ABB RAPID module: Module1.mod

MODULE Module1

! ## =========================================================================== ##
    ! MIT License
    ! Copyright (c) 2021 Roman Parak
    ! Permission is hereby granted, free of charge, to any person obtaining a copy
    ! of this software and associated documentation files (the "Software"), to deal
    ! in the Software without restriction, including without limitation the rights
    ! to use, copy, modify, merge, publish, distribute, sublicense, and/or sell
    ! copies of the Software, and to permit persons to whom the Software is
    ! furnished to do so, subject to the following conditions:
    ! The above copyright notice and this permission notice shall be included in all
    ! copies or substantial portions of the Software.
    ! THE SOFTWARE IS PROVIDED "AS IS", WITHOUT WARRANTY OF ANY KIND, EXPRESS OR
    ! IMPLIED, INCLUDING BUT NOT LIMITED TO THE WARRANTIES OF MERCHANTABILITY,
    ! FITNESS FOR A PARTICULAR PURPOSE AND NONINFRINGEMENT. IN NO EVENT SHALL THE
    ! AUTHORS OR COPYRIGHT HOLDERS BE LIABLE FOR ANY CLAIM, DAMAGES OR OTHER
    ! LIABILITY, WHETHER IN AN ACTION OF CONTRACT, TORT OR OTHERWISE, ARISING FROM,
    ! OUT OF OR IN CONNECTION WITH THE SOFTWARE OR THE USE OR OTHER DEALINGS IN THE
    ! SOFTWARE.
    ! ## =========================================================================== ##
    ! Author   : Roman Parak
    ! Email    : Roman.Parak@outlook.com
    ! Github   : https://github.com/rparak
    ! File Name: T_ROB1/Module1.mod
    ! ## =========================================================================== ##

    ! ############### EGM Initialization Parameters ############### !
    ! Identifier for the EGM correction.
     VAR robtarget starting_position;

    ! ################################## Externally Guided motion (EGM) - Main Cycle ################################## !
    PROC main()
        starting_position := CRobT(\Tool:=Tooldata_7\wobj:=wobj0);
        ConfJ\Off;
MoveJ RelTool (starting_position, 198, 1.3, -561 \Rx:=3.2, \Ry:=11.1, \Rz:=0), v200, z200, Tooldata_7;
MoveJ RelTool (starting_position, 198, 1.5, -561 \Rx:=3.1, \Ry:=11.1, \Rz:=0), v200, z200, Tooldata_7;
MoveJ RelTool (starting_position, 198, 1.7, -562 \Rx:=3, \Ry:=11.1, \Rz:=0), v200, z200, Tooldata_7;
MoveJ RelTool (starting_position, 198, 1.9, -562 \Rx:=2.8, \Ry:=11.1, \Rz:=0), v200, z200, Tooldata_7;
MoveJ RelTool (starting_position, 198, 2.1, -563 \Rx:=2.7, \Ry:=11.1, \Rz:=0), v200, z200, Tooldata_7;
MoveJ RelTool (starting_position, 198, 2.3, -563 \Rx:=2.6, \Ry:=11.1, \Rz:=0), v200, z200, Tooldata_7;
MoveJ RelTool (starting_position, 198, 2.6, -564 \Rx:=2.5, \Ry:=11.1, \Rz:=0), v200, z200, Tooldata_7;
MoveJ RelTool (starting_position, 197, 2.9, -565 \Rx:=2.3, \Ry:=11.1, \Rz:=0), v200, z200, Tooldata_7;
MoveJ RelTool (starting_position, 197, 3.1, -565 \Rx:=2.2, \Ry:=11.1, \Rz:=0), v200, z200, Tooldata_7;
MoveJ RelTool (starting_position, 197, 3.5, -566 \Rx:=2.1, \Ry:=10.8, \Rz:=0), v200, z200, Tooldata_7;
MoveJ RelTool (starting_position, 196, 3.8, -567 \Rx:=2, \Ry:=10.8, \Rz:=0), v200, z200, Tooldata_7;
MoveJ RelTool (starting_position, 196, 4.1, -567 \Rx:=2, \Ry:=10.8, \Rz:=0), v200, z200, Tooldata_7;
MoveJ RelTool (starting_position, 195, 4.5, -568 \Rx:=1.9, \Ry:=10.5, \Rz:=0), v200, z200, Tooldata_7;
MoveJ RelTool (starting_position, 195, 4.9, -569 \Rx:=1.9, \Ry:=10.5, \Rz:=0), v200, z200, Tooldata_7;
MoveJ RelTool (starting_position, 194, 5.3, -570 \Rx:=1.8, \Ry:=10.5, \Rz:=0), v200, z200, Tooldata_7;
MoveJ RelTool (starting_position, 194, 5.8, -571 \Rx:=1.8, \Ry:=10.5, \Rz:=0), v200, z200, Tooldata_7;
MoveJ RelTool (starting_position, 193, 6.3, -572 \Rx:=1.7, \Ry:=10.2, \Rz:=0), v200, z200, Tooldata_7;
MoveJ RelTool (starting_position, 192, 6.7, -573 \Rx:=1.7, \Ry:=10.2, \Rz:=0), v200, z200, Tooldata_7;
MoveJ RelTool (starting_position, 191, 7.3, -574 \Rx:=1.6, \Ry:=9.9, \Rz:=0), v200, z200, Tooldata_7;
MoveJ RelTool (starting_position, 190, 7.8, -575 \Rx:=1.6, \Ry:=9.9, \Rz:=0), v200, z200, Tooldata_7;
MoveJ RelTool (starting_position, 190, 8.4, -576 \Rx:=1.6, \Ry:=9.6, \Rz:=0), v200, z200, Tooldata_7;
MoveJ RelTool (starting_position, 189, 8.9, -577 \Rx:=1.5, \Ry:=9.6, \Rz:=0), v200, z200, Tooldata_7;
MoveJ RelTool (starting_position, 188, 9.6, -578 \Rx:=1.5, \Ry:=9.3, \Rz:=0), v200, z200, Tooldata_7;
MoveJ RelTool (starting_position, 187, 10.2, -579 \Rx:=1.5, \Ry:=9.3, \Rz:=0), v200, z200, Tooldata_7;
MoveJ RelTool (starting_position, 186, 10.8, -580 \Rx:=1.5, \Ry:=9, \Rz:=0), v200, z200, Tooldata_7;
MoveJ RelTool (starting_position, 185, 11.5, -581 \Rx:=1.5, \Ry:=8.7, \Rz:=0), v200, z200, Tooldata_7;
MoveJ RelTool (starting_position, 183, 12.1, -582 \Rx:=1.5, \Ry:=8.7, \Rz:=0), v200, z200, Tooldata_7;
MoveJ RelTool (starting_position, 182, 12.8, -583 \Rx:=1.5, \Ry:=8.4, \Rz:=0), v200, z200, Tooldata_7;
MoveJ RelTool (starting_position, 181, 13.5, -584 \Rx:=1.5, \Ry:=8.1, \Rz:=0), v200, z200, Tooldata_7;
MoveJ RelTool (starting_position, 179, 14.2, -585 \Rx:=1.5, \Ry:=7.8, \Rz:=0), v200, z200, Tooldata_7;
MoveJ RelTool (starting_position, 178, 14.9, -586 \Rx:=1.5, \Ry:=7.8, \Rz:=0), v200, z200, Tooldata_7;
MoveJ RelTool (starting_position, 177, 15.7, -586 \Rx:=1.5, \Ry:=7.5, \Rz:=0), v200, z200, Tooldata_7;
MoveJ RelTool (starting_position, 175, 16.4, -587 \Rx:=1.4, \Ry:=7.2, \Rz:=0), v200, z200, Tooldata_7;
MoveJ RelTool (starting_position, 174, 17.1, -588 \Rx:=1.4, \Ry:=6.9, \Rz:=0), v200, z200, Tooldata_7;
MoveJ RelTool (starting_position, 172, 17.8, -589 \Rx:=1.3, \Ry:=6.6, \Rz:=0), v200, z200, Tooldata_7;
MoveJ RelTool (starting_position, 171, 18.5, -589 \Rx:=1.3, \Ry:=6.3, \Rz:=0), v200, z200, Tooldata_7;
MoveJ RelTool (starting_position, 169, 19.2, -590 \Rx:=1.2, \Ry:=6, \Rz:=0), v200, z200, Tooldata_7;
MoveJ RelTool (starting_position, 168, 19.9, -591 \Rx:=1.1, \Ry:=6, \Rz:=0), v200, z200, Tooldata_7;
MoveJ RelTool (starting_position, 166, 20.5, -591 \Rx:=1, \Ry:=5.7, \Rz:=0), v200, z200, Tooldata_7;
MoveJ RelTool (starting_position, 165, 21.2, -592 \Rx:=0.9, \Ry:=5.4, \Rz:=0), v200, z200, Tooldata_7;
MoveJ RelTool (starting_position, 163, 21.8, -592 \Rx:=0.7, \Ry:=5.1, \Rz:=0), v200, z200, Tooldata_7;
MoveJ RelTool (starting_position, 162, 22.4, -593 \Rx:=0.6, \Ry:=4.8, \Rz:=0), v200, z200, Tooldata_7;
MoveJ RelTool (starting_position, 160, 23, -593 \Rx:=0.5, \Ry:=4.5, \Rz:=0), v200, z200, Tooldata_7;
MoveJ RelTool (starting_position, 158, 23.6, -594 \Rx:=0.4, \Ry:=4.2, \Rz:=0), v200, z200, Tooldata_7;
MoveJ RelTool (starting_position, 157, 24.1, -594 \Rx:=0.2, \Ry:=3.9, \Rz:=0), v200, z200, Tooldata_7;
MoveJ RelTool (starting_position, 155, 24.6, -594 \Rx:=0.1, \Ry:=3.6, \Rz:=0), v200, z200, Tooldata_7;
MoveJ RelTool (starting_position, 154, 25.1, -595 \Rx:=-0, \Ry:=3.6, \Rz:=0), v200, z200, Tooldata_7;
MoveJ RelTool (starting_position, 153, 25.6, -595 \Rx:=-0.1, \Ry:=3.3, \Rz:=0), v200, z200, Tooldata_7;
MoveJ RelTool (starting_position, 152, 26, -595 \Rx:=-0.1, \Ry:=3, \Rz:=0), v200, z200, Tooldata_7;
MoveJ RelTool (starting_position, 151, 26.4, -595 \Rx:=-0.2, \Ry:=3, \Rz:=0), v200, z200, Tooldata_7;
MoveJ RelTool (starting_position, 150, 26.8, -595 \Rx:=-0.3, \Ry:=2.7, \Rz:=0), v200, z200, Tooldata_7;
MoveJ RelTool (starting_position, 149, 27.1, -596 \Rx:=-0.3, \Ry:=2.7, \Rz:=0), v200, z200, Tooldata_7;
MoveJ RelTool (starting_position, 148, 27.5, -596 \Rx:=-0.3, \Ry:=2.4, \Rz:=0), v200, z200, Tooldata_7;
MoveJ RelTool (starting_position, 147, 27.8, -596 \Rx:=-0.3, \Ry:=2.1, \Rz:=0), v200, z200, Tooldata_7;
MoveJ RelTool (starting_position, 146, 28.2, -596 \Rx:=-0.3, \Ry:=2.1, \Rz:=0), v200, z200, Tooldata_7;
MoveJ RelTool (starting_position, 146, 28.5, -596 \Rx:=-0.3, \Ry:=2.1, \Rz:=0), v200, z200, Tooldata_7;
MoveJ RelTool (starting_position, 145, 28.8, -596 \Rx:=-0.3, \Ry:=2.1, \Rz:=0), v200, z200, Tooldata_7;
MoveJ RelTool (starting_position, 145, 29, -596 \Rx:=-0.2, \Ry:=1.8, \Rz:=0), v200, z200, Tooldata_7;
MoveJ RelTool (starting_position, 145, 29.3, -596 \Rx:=-0.1, \Ry:=1.8, \Rz:=0), v200, z200, Tooldata_7;
MoveJ RelTool (starting_position, 144, 29.6, -596 \Rx:=0, \Ry:=1.8, \Rz:=0), v200, z200, Tooldata_7;
MoveJ RelTool (starting_position, 144, 29.8, -596 \Rx:=0.1, \Ry:=1.8, \Rz:=0), v200, z200, Tooldata_7;
MoveJ RelTool (starting_position, 144, 30.1, -597 \Rx:=0.3, \Ry:=1.8, \Rz:=0), v200, z200, Tooldata_7;
MoveJ RelTool (starting_position, 144, 30.4, -597 \Rx:=0.4, \Ry:=1.8, \Rz:=0), v200, z200, Tooldata_7;
MoveJ RelTool (starting_position, 144, 30.6, -597 \Rx:=0.6, \Ry:=1.8, \Rz:=0), v200, z200, Tooldata_7;
MoveJ RelTool (starting_position, 144, 30.9, -597 \Rx:=0.8, \Ry:=1.8, \Rz:=0), v200, z200, Tooldata_7;
MoveJ RelTool (starting_position, 144, 31.2, -597 \Rx:=0.9, \Ry:=1.8, \Rz:=0), v200, z200, Tooldata_7;
MoveJ RelTool (starting_position, 144, 31.5, -597 \Rx:=1.2, \Ry:=1.8, \Rz:=0), v200, z200, Tooldata_7;
MoveJ RelTool (starting_position, 144, 31.8, -597 \Rx:=1.4, \Ry:=1.8, \Rz:=0), v200, z200, Tooldata_7;
MoveJ RelTool (starting_position, 144, 32.1, -597 \Rx:=1.7, \Ry:=1.8, \Rz:=0), v200, z200, Tooldata_7;
MoveJ RelTool (starting_position, 145, 32.4, -597 \Rx:=2, \Ry:=1.8, \Rz:=0), v200, z200, Tooldata_7;
MoveJ RelTool (starting_position, 145, 32.8, -597 \Rx:=2.4, \Ry:=1.8, \Rz:=0), v200, z200, Tooldata_7;
MoveJ RelTool (starting_position, 145, 33.2, -597 \Rx:=2.7, \Ry:=2.1, \Rz:=0), v200, z200, Tooldata_7;
MoveJ RelTool (starting_position, 146, 33.6, -597 \Rx:=3.1, \Ry:=2.1, \Rz:=0), v200, z200, Tooldata_7;
MoveJ RelTool (starting_position, 146, 34, -598 \Rx:=3.4, \Ry:=2.1, \Rz:=0), v200, z200, Tooldata_7;
MoveJ RelTool (starting_position, 147, 34.4, -598 \Rx:=3.7, \Ry:=2.4, \Rz:=0), v200, z200, Tooldata_7;
MoveJ RelTool (starting_position, 147, 34.8, -598 \Rx:=4.1, \Ry:=2.4, \Rz:=0), v200, z200, Tooldata_7;
MoveJ RelTool (starting_position, 148, 35.3, -598 \Rx:=4.4, \Ry:=2.4, \Rz:=0), v200, z200, Tooldata_7;
MoveJ RelTool (starting_position, 148, 35.9, -598 \Rx:=4.7, \Ry:=2.4, \Rz:=0), v200, z200, Tooldata_7;
MoveJ RelTool (starting_position, 149, 36.4, -599 \Rx:=5, \Ry:=2.7, \Rz:=0), v200, z200, Tooldata_7;
MoveJ RelTool (starting_position, 149, 37, -599 \Rx:=5.3, \Ry:=2.7, \Rz:=0), v200, z200, Tooldata_7;
MoveJ RelTool (starting_position, 150, 37.6, -599 \Rx:=5.6, \Ry:=2.7, \Rz:=0), v200, z200, Tooldata_7;
MoveJ RelTool (starting_position, 150, 38.2, -600 \Rx:=5.8, \Ry:=3, \Rz:=0), v200, z200, Tooldata_7;
MoveJ RelTool (starting_position, 151, 38.8, -600 \Rx:=5.9, \Ry:=3, \Rz:=0), v200, z200, Tooldata_7;
MoveJ RelTool (starting_position, 151, 39.5, -600 \Rx:=6.1, \Ry:=3, \Rz:=0), v200, z200, Tooldata_7;
MoveJ RelTool (starting_position, 151, 40.2, -601 \Rx:=6.2, \Ry:=3, \Rz:=0), v200, z200, Tooldata_7;
MoveJ RelTool (starting_position, 151, 40.9, -601 \Rx:=6.3, \Ry:=3, \Rz:=0), v200, z200, Tooldata_7;
MoveJ RelTool (starting_position, 152, 41.6, -602 \Rx:=6.3, \Ry:=3, \Rz:=0), v200, z200, Tooldata_7;
MoveJ RelTool (starting_position, 152, 42.4, -602 \Rx:=6.2, \Ry:=3.3, \Rz:=0), v200, z200, Tooldata_7;
MoveJ RelTool (starting_position, 152, 43.1, -603 \Rx:=6.2, \Ry:=3.3, \Rz:=0), v200, z200, Tooldata_7;
MoveJ RelTool (starting_position, 153, 43.8, -603 \Rx:=6, \Ry:=3.3, \Rz:=0), v200, z200, Tooldata_7;
MoveJ RelTool (starting_position, 153, 44.6, -604 \Rx:=5.9, \Ry:=3.3, \Rz:=0), v200, z200, Tooldata_7;
MoveJ RelTool (starting_position, 153, 45.4, -604 \Rx:=5.7, \Ry:=3.3, \Rz:=0), v200, z200, Tooldata_7;
MoveJ RelTool (starting_position, 153, 46.1, -605 \Rx:=5.6, \Ry:=3.6, \Rz:=0), v200, z200, Tooldata_7;
MoveJ RelTool (starting_position, 153, 46.9, -605 \Rx:=5.3, \Ry:=3.3, \Rz:=0), v200, z200, Tooldata_7;
MoveJ RelTool (starting_position, 153, 47.6, -606 \Rx:=5.1, \Ry:=3.3, \Rz:=0), v200, z200, Tooldata_7;
MoveJ RelTool (starting_position, 153, 48.3, -606 \Rx:=4.9, \Ry:=3.3, \Rz:=0), v200, z200, Tooldata_7;
MoveJ RelTool (starting_position, 152, 49.1, -606 \Rx:=4.7, \Ry:=3.3, \Rz:=0), v200, z200, Tooldata_7;
MoveJ RelTool (starting_position, 152, 49.8, -607 \Rx:=4.5, \Ry:=3.3, \Rz:=0), v200, z200, Tooldata_7;
MoveJ RelTool (starting_position, 152, 50.5, -607 \Rx:=4.2, \Ry:=3, \Rz:=0), v200, z200, Tooldata_7;
MoveJ RelTool (starting_position, 151, 51.1, -608 \Rx:=4, \Ry:=3, \Rz:=0), v200, z200, Tooldata_7;
MoveJ RelTool (starting_position, 151, 51.8, -608 \Rx:=3.9, \Ry:=3, \Rz:=0), v200, z200, Tooldata_7;
MoveJ RelTool (starting_position, 151, 52.4, -608 \Rx:=3.7, \Ry:=3, \Rz:=0), v200, z200, Tooldata_7;
MoveJ RelTool (starting_position, 150, 53, -609 \Rx:=3.6, \Ry:=3, \Rz:=0), v200, z200, Tooldata_7;
MoveJ RelTool (starting_position, 150, 53.6, -609 \Rx:=3.5, \Ry:=2.7, \Rz:=0), v200, z200, Tooldata_7;
MoveJ RelTool (starting_position, 150, 54.1, -609 \Rx:=3.4, \Ry:=2.7, \Rz:=0), v200, z200, Tooldata_7;
MoveJ RelTool (starting_position, 149, 54.6, -609 \Rx:=3.4, \Ry:=2.7, \Rz:=0), v200, z200, Tooldata_7;
MoveJ RelTool (starting_position, 149, 55.1, -610 \Rx:=3.3, \Ry:=2.7, \Rz:=0), v200, z200, Tooldata_7;
MoveJ RelTool (starting_position, 148, 55.6, -610 \Rx:=3.3, \Ry:=2.4, \Rz:=0), v200, z200, Tooldata_7;
MoveJ RelTool (starting_position, 148, 56, -610 \Rx:=3.4, \Ry:=2.4, \Rz:=0), v200, z200, Tooldata_7;
MoveJ RelTool (starting_position, 147, 56.4, -610 \Rx:=3.4, \Ry:=2.4, \Rz:=0), v200, z200, Tooldata_7;
MoveJ RelTool (starting_position, 147, 56.8, -610 \Rx:=3.6, \Ry:=2.1, \Rz:=0), v200, z200, Tooldata_7;
MoveJ RelTool (starting_position, 146, 57.1, -610 \Rx:=3.7, \Ry:=2.1, \Rz:=0), v200, z200, Tooldata_7;
MoveJ RelTool (starting_position, 146, 57.5, -611 \Rx:=4, \Ry:=2.1, \Rz:=0), v200, z200, Tooldata_7;
MoveJ RelTool (starting_position, 145, 57.8, -611 \Rx:=4.2, \Ry:=2.1, \Rz:=0), v200, z200, Tooldata_7;
MoveJ RelTool (starting_position, 145, 58.1, -611 \Rx:=4.6, \Ry:=1.8, \Rz:=0), v200, z200, Tooldata_7;
MoveJ RelTool (starting_position, 144, 58.4, -611 \Rx:=5, \Ry:=1.8, \Rz:=0), v200, z200, Tooldata_7;
MoveJ RelTool (starting_position, 144, 58.7, -611 \Rx:=5.4, \Ry:=1.8, \Rz:=0), v200, z200, Tooldata_7;
MoveJ RelTool (starting_position, 143, 59, -612 \Rx:=5.8, \Ry:=1.5, \Rz:=0), v200, z200, Tooldata_7;
MoveJ RelTool (starting_position, 142, 59.2, -612 \Rx:=6.2, \Ry:=1.5, \Rz:=0), v200, z200, Tooldata_7;
MoveJ RelTool (starting_position, 142, 59.5, -612 \Rx:=6.6, \Ry:=1.5, \Rz:=0), v200, z200, Tooldata_7;
MoveJ RelTool (starting_position, 141, 59.7, -612 \Rx:=7.1, \Ry:=1.2, \Rz:=0), v200, z200, Tooldata_7;
MoveJ RelTool (starting_position, 140, 60, -612 \Rx:=7.6, \Ry:=1.2, \Rz:=0), v200, z200, Tooldata_7;
MoveJ RelTool (starting_position, 139, 60.2, -613 \Rx:=8.1, \Ry:=0.9, \Rz:=0), v200, z200, Tooldata_7;
MoveJ RelTool (starting_position, 139, 60.5, -613 \Rx:=8.5, \Ry:=0.9, \Rz:=0), v200, z200, Tooldata_7;
MoveJ RelTool (starting_position, 138, 60.7, -613 \Rx:=9, \Ry:=0.6, \Rz:=0), v200, z200, Tooldata_7;
MoveJ RelTool (starting_position, 137, 61, -613 \Rx:=9.4, \Ry:=0.6, \Rz:=0), v200, z200, Tooldata_7;
MoveJ RelTool (starting_position, 136, 61.2, -613 \Rx:=9.8, \Ry:=0.6, \Rz:=0), v200, z200, Tooldata_7;
MoveJ RelTool (starting_position, 135, 61.5, -614 \Rx:=10.1, \Ry:=0.3, \Rz:=0), v200, z200, Tooldata_7;
MoveJ RelTool (starting_position, 134, 61.8, -614 \Rx:=10.3, \Ry:=0, \Rz:=0), v200, z200, Tooldata_7;
MoveJ RelTool (starting_position, 133, 62.1, -614 \Rx:=10.5, \Ry:=-0, \Rz:=0), v200, z200, Tooldata_7;
MoveJ RelTool (starting_position, 133, 62.5, -614 \Rx:=10.6, \Ry:=-0.3, \Rz:=0), v200, z200, Tooldata_7;
MoveJ RelTool (starting_position, 132, 62.8, -614 \Rx:=10.6, \Ry:=-0.3, \Rz:=0), v200, z200, Tooldata_7;
MoveJ RelTool (starting_position, 131, 63.2, -614 \Rx:=10.6, \Ry:=-0.6, \Rz:=0), v200, z200, Tooldata_7;
MoveJ RelTool (starting_position, 130, 63.6, -614 \Rx:=10.4, \Ry:=-0.6, \Rz:=0), v200, z200, Tooldata_7;
MoveJ RelTool (starting_position, 129, 64, -614 \Rx:=10.1, \Ry:=-0.9, \Rz:=0), v200, z200, Tooldata_7;
MoveJ RelTool (starting_position, 128, 64.4, -614 \Rx:=9.8, \Ry:=-1.2, \Rz:=0), v200, z200, Tooldata_7;
MoveJ RelTool (starting_position, 127, 64.8, -614 \Rx:=9.5, \Ry:=-1.2, \Rz:=0), v200, z200, Tooldata_7;
MoveJ RelTool (starting_position, 126, 65.3, -614 \Rx:=9.1, \Ry:=-1.5, \Rz:=0), v200, z200, Tooldata_7;
MoveJ RelTool (starting_position, 125, 65.9, -613 \Rx:=8.7, \Ry:=-1.5, \Rz:=0), v200, z200, Tooldata_7;
MoveJ RelTool (starting_position, 124, 66.4, -613 \Rx:=8.2, \Ry:=-1.8, \Rz:=0), v200, z200, Tooldata_7;
MoveJ RelTool (starting_position, 123, 67, -613 \Rx:=7.7, \Ry:=-1.8, \Rz:=0), v200, z200, Tooldata_7;
MoveJ RelTool (starting_position, 122, 67.6, -613 \Rx:=7.2, \Ry:=-2.1, \Rz:=0), v200, z200, Tooldata_7;
MoveJ RelTool (starting_position, 122, 68.2, -612 \Rx:=6.7, \Ry:=-2.1, \Rz:=0), v200, z200, Tooldata_7;
MoveJ RelTool (starting_position, 121, 68.8, -612 \Rx:=6.2, \Ry:=-2.1, \Rz:=0), v200, z200, Tooldata_7;
MoveJ RelTool (starting_position, 120, 69.5, -612 \Rx:=5.7, \Ry:=-2.4, \Rz:=0), v200, z200, Tooldata_7;
MoveJ RelTool (starting_position, 119, 70.2, -611 \Rx:=5.2, \Ry:=-2.7, \Rz:=0), v200, z200, Tooldata_7;
MoveJ RelTool (starting_position, 118, 70.9, -611 \Rx:=4.8, \Ry:=-2.7, \Rz:=0), v200, z200, Tooldata_7;
MoveJ RelTool (starting_position, 117, 71.6, -611 \Rx:=4.4, \Ry:=-3, \Rz:=0), v200, z200, Tooldata_7;
MoveJ RelTool (starting_position, 116, 72.4, -610 \Rx:=4.1, \Ry:=-3, \Rz:=0), v200, z200, Tooldata_7;
MoveJ RelTool (starting_position, 116, 73.1, -610 \Rx:=3.8, \Ry:=-3, \Rz:=0), v200, z200, Tooldata_7;
MoveJ RelTool (starting_position, 115, 73.8, -610 \Rx:=3.5, \Ry:=-3.3, \Rz:=0), v200, z200, Tooldata_7;
MoveJ RelTool (starting_position, 114, 74.6, -609 \Rx:=3.3, \Ry:=-3.3, \Rz:=0), v200, z200, Tooldata_7;
MoveJ RelTool (starting_position, 114, 75.4, -609 \Rx:=3.1, \Ry:=-3.6, \Rz:=0), v200, z200, Tooldata_7;
MoveJ RelTool (starting_position, 113, 76.1, -608 \Rx:=3, \Ry:=-3.6, \Rz:=0), v200, z200, Tooldata_7;
MoveJ RelTool (starting_position, 113, 76.9, -608 \Rx:=3, \Ry:=-3.6, \Rz:=0), v200, z200, Tooldata_7;
MoveJ RelTool (starting_position, 113, 77.6, -608 \Rx:=2.9, \Ry:=-3.6, \Rz:=0), v200, z200, Tooldata_7;
MoveJ RelTool (starting_position, 112, 78.3, -607 \Rx:=2.9, \Ry:=-3.6, \Rz:=0), v200, z200, Tooldata_7;
MoveJ RelTool (starting_position, 112, 79.1, -607 \Rx:=2.9, \Ry:=-3.9, \Rz:=0), v200, z200, Tooldata_7;
MoveJ RelTool (starting_position, 111, 79.8, -606 \Rx:=2.9, \Ry:=-3.9, \Rz:=0), v200, z200, Tooldata_7;
MoveJ RelTool (starting_position, 111, 80.5, -606 \Rx:=3, \Ry:=-3.9, \Rz:=0), v200, z200, Tooldata_7;
MoveJ RelTool (starting_position, 110, 81.1, -605 \Rx:=3.1, \Ry:=-4.2, \Rz:=0), v200, z200, Tooldata_7;
MoveJ RelTool (starting_position, 110, 81.8, -605 \Rx:=3.1, \Ry:=-4.2, \Rz:=0), v200, z200, Tooldata_7;
MoveJ RelTool (starting_position, 110, 82.4, -605 \Rx:=3.2, \Ry:=-4.2, \Rz:=0), v200, z200, Tooldata_7;
MoveJ RelTool (starting_position, 109, 83, -604 \Rx:=3.2, \Ry:=-4.2, \Rz:=0), v200, z200, Tooldata_7;
MoveJ RelTool (starting_position, 109, 83.6, -604 \Rx:=3.2, \Ry:=-4.2, \Rz:=0), v200, z200, Tooldata_7;
MoveJ RelTool (starting_position, 108, 84.1, -603 \Rx:=3.3, \Ry:=-4.5, \Rz:=0), v200, z200, Tooldata_7;
MoveJ RelTool (starting_position, 108, 84.6, -603 \Rx:=3.3, \Ry:=-4.5, \Rz:=0), v200, z200, Tooldata_7;
MoveJ RelTool (starting_position, 108, 85.1, -602 \Rx:=3.3, \Ry:=-4.5, \Rz:=0), v200, z200, Tooldata_7;
MoveJ RelTool (starting_position, 107, 85.6, -602 \Rx:=3.3, \Ry:=-4.5, \Rz:=0), v200, z200, Tooldata_7;
MoveJ RelTool (starting_position, 107, 86, -602 \Rx:=3.3, \Ry:=-4.8, \Rz:=0), v200, z200, Tooldata_7;
MoveJ RelTool (starting_position, 106, 86.4, -601 \Rx:=3.3, \Ry:=-4.8, \Rz:=0), v200, z200, Tooldata_7;
MoveJ RelTool (starting_position, 106, 86.8, -601 \Rx:=3.2, \Ry:=-4.8, \Rz:=0), v200, z200, Tooldata_7;
MoveJ RelTool (starting_position, 106, 87.1, -600 \Rx:=3.2, \Ry:=-4.8, \Rz:=0), v200, z200, Tooldata_7;
MoveJ RelTool (starting_position, 106, 87.5, -600 \Rx:=3.2, \Ry:=-4.8, \Rz:=0), v200, z200, Tooldata_7;
MoveJ RelTool (starting_position, 106, 87.7, -600 \Rx:=3.1, \Ry:=-4.8, \Rz:=0), v200, z200, Tooldata_7;
MoveJ RelTool (starting_position, 105, 88, -599 \Rx:=3.1, \Ry:=-5.1, \Rz:=0), v200, z200, Tooldata_7;
MoveJ RelTool (starting_position, 105, 88.3, -599 \Rx:=3.1, \Ry:=-5.1, \Rz:=0), v200, z200, Tooldata_7;
MoveJ RelTool (starting_position, 105, 88.6, -598 \Rx:=3, \Ry:=-4.8, \Rz:=0), v200, z200, Tooldata_7;
MoveJ RelTool (starting_position, 105, 88.8, -598 \Rx:=3, \Ry:=-4.8, \Rz:=0), v200, z200, Tooldata_7;
MoveJ RelTool (starting_position, 105, 89.1, -597 \Rx:=3, \Ry:=-5.1, \Rz:=0), v200, z200, Tooldata_7;
MoveJ RelTool (starting_position, 105, 89.3, -597 \Rx:=3, \Ry:=-5.1, \Rz:=0), v200, z200, Tooldata_7;
MoveJ RelTool (starting_position, 104, 89.5, -596 \Rx:=2.9, \Ry:=-5.1, \Rz:=0), v200, z200, Tooldata_7;
MoveJ RelTool (starting_position, 104, 89.7, -595 \Rx:=2.9, \Ry:=-5.1, \Rz:=0), v200, z200, Tooldata_7;
MoveJ RelTool (starting_position, 104, 90, -595 \Rx:=2.8, \Ry:=-5.1, \Rz:=0), v200, z200, Tooldata_7;
MoveJ RelTool (starting_position, 105, 90.2, -594 \Rx:=2.7, \Ry:=-5.1, \Rz:=0), v200, z200, Tooldata_7;
MoveJ RelTool (starting_position, 105, 90.4, -594 \Rx:=2.6, \Ry:=-5.1, \Rz:=0), v200, z200, Tooldata_7;
MoveJ RelTool (starting_position, 105, 90.6, -593 \Rx:=2.4, \Ry:=-4.8, \Rz:=0), v200, z200, Tooldata_7;
MoveJ RelTool (starting_position, 106, 90.9, -592 \Rx:=2.3, \Ry:=-4.8, \Rz:=0), v200, z200, Tooldata_7;
MoveJ RelTool (starting_position, 106, 91.1, -592 \Rx:=2.1, \Ry:=-4.8, \Rz:=0), v200, z200, Tooldata_7;
MoveJ RelTool (starting_position, 107, 91.4, -591 \Rx:=1.9, \Ry:=-4.8, \Rz:=0), v200, z200, Tooldata_7;
MoveJ RelTool (starting_position, 107, 91.6, -590 \Rx:=1.7, \Ry:=-4.5, \Rz:=0), v200, z200, Tooldata_7;
MoveJ RelTool (starting_position, 108, 91.9, -590 \Rx:=1.5, \Ry:=-4.5, \Rz:=0), v200, z200, Tooldata_7;
MoveJ RelTool (starting_position, 108, 92.2, -589 \Rx:=1.3, \Ry:=-4.5, \Rz:=0), v200, z200, Tooldata_7;
MoveJ RelTool (starting_position, 109, 92.5, -588 \Rx:=1.1, \Ry:=-4.2, \Rz:=0), v200, z200, Tooldata_7;
MoveJ RelTool (starting_position, 110, 92.8, -588 \Rx:=0.9, \Ry:=-4.2, \Rz:=0), v200, z200, Tooldata_7;
MoveJ RelTool (starting_position, 111, 93.2, -587 \Rx:=0.7, \Ry:=-3.9, \Rz:=0), v200, z200, Tooldata_7;
MoveJ RelTool (starting_position, 112, 93.6, -587 \Rx:=0.4, \Ry:=-3.9, \Rz:=0), v200, z200, Tooldata_7;
MoveJ RelTool (starting_position, 113, 94, -586 \Rx:=0.2, \Ry:=-3.6, \Rz:=0), v200, z200, Tooldata_7;
MoveJ RelTool (starting_position, 114, 94.4, -586 \Rx:=0, \Ry:=-3.6, \Rz:=0), v200, z200, Tooldata_7;
MoveJ RelTool (starting_position, 115, 94.8, -585 \Rx:=-0.2, \Ry:=-3.3, \Rz:=0), v200, z200, Tooldata_7;
MoveJ RelTool (starting_position, 116, 95.3, -585 \Rx:=-0.4, \Ry:=-3, \Rz:=0), v200, z200, Tooldata_7;
MoveJ RelTool (starting_position, 117, 95.9, -584 \Rx:=-0.5, \Ry:=-2.7, \Rz:=0), v200, z200, Tooldata_7;
MoveJ RelTool (starting_position, 119, 96.4, -584 \Rx:=-0.7, \Ry:=-2.7, \Rz:=0), v200, z200, Tooldata_7;
MoveJ RelTool (starting_position, 120, 97, -584 \Rx:=-0.8, \Ry:=-2.4, \Rz:=0), v200, z200, Tooldata_7;
MoveJ RelTool (starting_position, 122, 97.6, -583 \Rx:=-0.9, \Ry:=-2.1, \Rz:=0), v200, z200, Tooldata_7;
MoveJ RelTool (starting_position, 123, 98.2, -583 \Rx:=-1, \Ry:=-1.8, \Rz:=0), v200, z200, Tooldata_7;
MoveJ RelTool (starting_position, 125, 98.8, -583 \Rx:=-1, \Ry:=-1.5, \Rz:=0), v200, z200, Tooldata_7;
MoveJ RelTool (starting_position, 126, 99.5, -583 \Rx:=-1, \Ry:=-1.2, \Rz:=0), v200, z200, Tooldata_7;
MoveJ RelTool (starting_position, 127, 100.2, -583 \Rx:=-1, \Ry:=-1.2, \Rz:=0), v200, z200, Tooldata_7;
MoveJ RelTool (starting_position, 129, 100.9, -583 \Rx:=-0.9, \Ry:=-0.9, \Rz:=0), v200, z200, Tooldata_7;
MoveJ RelTool (starting_position, 130, 101.6, -583 \Rx:=-0.8, \Ry:=-0.6, \Rz:=0), v200, z200, Tooldata_7;
MoveJ RelTool (starting_position, 132, 102.4, -583 \Rx:=-0.7, \Ry:=-0.3, \Rz:=0), v200, z200, Tooldata_7;
MoveJ RelTool (starting_position, 133, 103.1, -583 \Rx:=-0.6, \Ry:=-0, \Rz:=0), v200, z200, Tooldata_7;
MoveJ RelTool (starting_position, 135, 103.8, -583 \Rx:=-0.4, \Ry:=0.3, \Rz:=0), v200, z200, Tooldata_7;
MoveJ RelTool (starting_position, 136, 104.6, -583 \Rx:=-0.3, \Ry:=0.3, \Rz:=0), v200, z200, Tooldata_7;
MoveJ RelTool (starting_position, 137, 105.4, -583 \Rx:=-0.1, \Ry:=0.6, \Rz:=0), v200, z200, Tooldata_7;
MoveJ RelTool (starting_position, 139, 106.1, -583 \Rx:=0.1, \Ry:=0.9, \Rz:=0), v200, z200, Tooldata_7;
MoveJ RelTool (starting_position, 140, 106.9, -584 \Rx:=0.3, \Ry:=1.2, \Rz:=0), v200, z200, Tooldata_7;
MoveJ RelTool (starting_position, 141, 107.6, -584 \Rx:=0.5, \Ry:=1.2, \Rz:=0), v200, z200, Tooldata_7;
MoveJ RelTool (starting_position, 143, 108.3, -584 \Rx:=0.7, \Ry:=1.5, \Rz:=0), v200, z200, Tooldata_7;
MoveJ RelTool (starting_position, 144, 109.1, -584 \Rx:=0.9, \Ry:=1.8, \Rz:=0), v200, z200, Tooldata_7;
MoveJ RelTool (starting_position, 145, 109.8, -585 \Rx:=1.1, \Ry:=2.1, \Rz:=0), v200, z200, Tooldata_7;
MoveJ RelTool (starting_position, 146, 110.5, -585 \Rx:=1.3, \Ry:=2.1, \Rz:=0), v200, z200, Tooldata_7;
MoveJ RelTool (starting_position, 147, 111.1, -585 \Rx:=1.4, \Ry:=2.4, \Rz:=0), v200, z200, Tooldata_7;
MoveJ RelTool (starting_position, 148, 111.8, -585 \Rx:=1.6, \Ry:=2.4, \Rz:=0), v200, z200, Tooldata_7;
MoveJ RelTool (starting_position, 150, 112.4, -585 \Rx:=1.8, \Ry:=2.7, \Rz:=0), v200, z200, Tooldata_7;
MoveJ RelTool (starting_position, 151, 113, -586 \Rx:=1.9, \Ry:=3, \Rz:=0), v200, z200, Tooldata_7;
MoveJ RelTool (starting_position, 152, 113.6, -586 \Rx:=2.1, \Ry:=3.3, \Rz:=0), v200, z200, Tooldata_7;
MoveJ RelTool (starting_position, 153, 114.1, -586 \Rx:=2.3, \Ry:=3.3, \Rz:=0), v200, z200, Tooldata_7;
MoveJ RelTool (starting_position, 155, 114.6, -586 \Rx:=2.5, \Ry:=3.6, \Rz:=0), v200, z200, Tooldata_7;
MoveJ RelTool (starting_position, 156, 115.1, -587 \Rx:=2.6, \Ry:=3.9, \Rz:=0), v200, z200, Tooldata_7;
MoveJ RelTool (starting_position, 157, 115.6, -587 \Rx:=2.8, \Ry:=4.2, \Rz:=0), v200, z200, Tooldata_7;
MoveJ RelTool (starting_position, 158, 116, -587 \Rx:=3, \Ry:=4.2, \Rz:=0), v200, z200, Tooldata_7;
MoveJ RelTool (starting_position, 159, 116.4, -588 \Rx:=3.1, \Ry:=4.2, \Rz:=0), v200, z200, Tooldata_7;
MoveJ RelTool (starting_position, 159, 116.8, -588 \Rx:=3.2, \Ry:=4.5, \Rz:=0), v200, z200, Tooldata_7;
MoveJ RelTool (starting_position, 160, 117.1, -589 \Rx:=3.4, \Ry:=4.5, \Rz:=0), v200, z200, Tooldata_7;
MoveJ RelTool (starting_position, 161, 117.5, -589 \Rx:=3.5, \Ry:=4.8, \Rz:=0), v200, z200, Tooldata_7;
MoveJ RelTool (starting_position, 161, 117.7, -590 \Rx:=3.6, \Ry:=4.8, \Rz:=0), v200, z200, Tooldata_7;
MoveJ RelTool (starting_position, 162, 118, -590 \Rx:=3.7, \Ry:=4.8, \Rz:=0), v200, z200, Tooldata_7;
MoveJ RelTool (starting_position, 162, 118.3, -591 \Rx:=3.8, \Ry:=5.1, \Rz:=0), v200, z200, Tooldata_7;
MoveJ RelTool (starting_position, 163, 118.5, -591 \Rx:=3.9, \Ry:=5.1, \Rz:=0), v200, z200, Tooldata_7;
MoveJ RelTool (starting_position, 163, 118.7, -592 \Rx:=4, \Ry:=5.1, \Rz:=0), v200, z200, Tooldata_7;
MoveJ RelTool (starting_position, 163, 119, -593 \Rx:=4, \Ry:=5.1, \Rz:=0), v200, z200, Tooldata_7;
MoveJ RelTool (starting_position, 163, 119.2, -593 \Rx:=4.1, \Ry:=5.1, \Rz:=0), v200, z200, Tooldata_7;
MoveJ RelTool (starting_position, 163, 119.4, -594 \Rx:=4.2, \Ry:=5.1, \Rz:=0), v200, z200, Tooldata_7;
MoveJ RelTool (starting_position, 162, 119.6, -595 \Rx:=4.3, \Ry:=5.1, \Rz:=0), v200, z200, Tooldata_7;
MoveJ RelTool (starting_position, 162, 119.8, -596 \Rx:=4.4, \Ry:=4.8, \Rz:=0), v200, z200, Tooldata_7;
MoveJ RelTool (starting_position, 161, 120, -596 \Rx:=4.4, \Ry:=4.8, \Rz:=0), v200, z200, Tooldata_7;
MoveJ RelTool (starting_position, 160, 120.2, -597 \Rx:=4.4, \Ry:=4.5, \Rz:=0), v200, z200, Tooldata_7;
MoveJ RelTool (starting_position, 160, 120.4, -598 \Rx:=4.4, \Ry:=4.5, \Rz:=0), v200, z200, Tooldata_7;
MoveJ RelTool (starting_position, 159, 120.6, -599 \Rx:=4.4, \Ry:=4.5, \Rz:=0), v200, z200, Tooldata_7;
MoveJ RelTool (starting_position, 158, 120.8, -600 \Rx:=4.4, \Ry:=4.2, \Rz:=0), v200, z200, Tooldata_7;
MoveJ RelTool (starting_position, 156, 121, -600 \Rx:=4.3, \Ry:=3.9, \Rz:=0), v200, z200, Tooldata_7;
MoveJ RelTool (starting_position, 155, 121.2, -601 \Rx:=4.2, \Ry:=3.6, \Rz:=0), v200, z200, Tooldata_7;
MoveJ RelTool (starting_position, 154, 121.4, -602 \Rx:=4.1, \Ry:=3.6, \Rz:=0), v200, z200, Tooldata_7;
MoveJ RelTool (starting_position, 152, 121.7, -602 \Rx:=4, \Ry:=3.3, \Rz:=0), v200, z200, Tooldata_7;
MoveJ RelTool (starting_position, 151, 121.9, -603 \Rx:=3.7, \Ry:=3, \Rz:=0), v200, z200, Tooldata_7;
MoveJ RelTool (starting_position, 149, 122.2, -604 \Rx:=3.5, \Ry:=2.7, \Rz:=0), v200, z200, Tooldata_7;
MoveJ RelTool (starting_position, 148, 122.5, -604 \Rx:=3.2, \Ry:=2.4, \Rz:=0), v200, z200, Tooldata_7;
MoveJ RelTool (starting_position, 146, 122.8, -605 \Rx:=2.8, \Ry:=2.1, \Rz:=0), v200, z200, Tooldata_7;
MoveJ RelTool (starting_position, 144, 123.2, -605 \Rx:=2.4, \Ry:=1.8, \Rz:=0), v200, z200, Tooldata_7;
MoveJ RelTool (starting_position, 142, 123.6, -605 \Rx:=2, \Ry:=1.5, \Rz:=0), v200, z200, Tooldata_7;
MoveJ RelTool (starting_position, 140, 124, -606 \Rx:=1.6, \Ry:=0.9, \Rz:=0), v200, z200, Tooldata_7;
MoveJ RelTool (starting_position, 138, 124.4, -606 \Rx:=1.1, \Ry:=0.6, \Rz:=0), v200, z200, Tooldata_7;
MoveJ RelTool (starting_position, 136, 124.8, -606 \Rx:=0.6, \Ry:=0.6, \Rz:=0), v200, z200, Tooldata_7;
MoveJ RelTool (starting_position, 135, 125.3, -606 \Rx:=0.1, \Ry:=0.3, \Rz:=0), v200, z200, Tooldata_7;
MoveJ RelTool (starting_position, 133, 125.9, -606 \Rx:=-0.5, \Ry:=-0.3, \Rz:=0), v200, z200, Tooldata_7;
MoveJ RelTool (starting_position, 131, 126.4, -606 \Rx:=-1.1, \Ry:=-0.6, \Rz:=0), v200, z200, Tooldata_7;
MoveJ RelTool (starting_position, 128, 127, -605 \Rx:=-1.7, \Ry:=-0.9, \Rz:=0), v200, z200, Tooldata_7;
MoveJ RelTool (starting_position, 126, 127.6, -605 \Rx:=-2.3, \Ry:=-1.2, \Rz:=0), v200, z200, Tooldata_7;
MoveJ RelTool (starting_position, 124, 128.2, -605 \Rx:=-2.8, \Ry:=-1.8, \Rz:=0), v200, z200, Tooldata_7;
MoveJ RelTool (starting_position, 122, 128.8, -604 \Rx:=-3.4, \Ry:=-2.1, \Rz:=0), v200, z200, Tooldata_7;
MoveJ RelTool (starting_position, 119, 129.5, -604 \Rx:=-4, \Ry:=-2.4, \Rz:=0), v200, z200, Tooldata_7;
MoveJ RelTool (starting_position, 117, 130.2, -603 \Rx:=-4.5, \Ry:=-3, \Rz:=0), v200, z200, Tooldata_7;
MoveJ RelTool (starting_position, 115, 130.9, -602 \Rx:=-5, \Ry:=-3.3, \Rz:=0), v200, z200, Tooldata_7;
MoveJ RelTool (starting_position, 113, 131.6, -602 \Rx:=-5.5, \Ry:=-3.6, \Rz:=0), v200, z200, Tooldata_7;
MoveJ RelTool (starting_position, 111, 132.4, -601 \Rx:=-5.9, \Ry:=-3.9, \Rz:=0), v200, z200, Tooldata_7;
MoveJ RelTool (starting_position, 109, 133.1, -600 \Rx:=-6.3, \Ry:=-4.5, \Rz:=0), v200, z200, Tooldata_7;
MoveJ RelTool (starting_position, 106, 133.8, -599 \Rx:=-6.7, \Ry:=-4.8, \Rz:=0), v200, z200, Tooldata_7;
MoveJ RelTool (starting_position, 104, 134.6, -599 \Rx:=-6.9, \Ry:=-5.1, \Rz:=0), v200, z200, Tooldata_7;
MoveJ RelTool (starting_position, 102, 135.4, -598 \Rx:=-7.2, \Ry:=-5.4, \Rz:=0), v200, z200, Tooldata_7;
MoveJ RelTool (starting_position, 100, 136.1, -597 \Rx:=-7.3, \Ry:=-5.7, \Rz:=0), v200, z200, Tooldata_7;
MoveJ RelTool (starting_position, 98, 136.9, -597 \Rx:=-7.4, \Ry:=-6.3, \Rz:=0), v200, z200, Tooldata_7;
MoveJ RelTool (starting_position, 95, 137.6, -596 \Rx:=-7.4, \Ry:=-6.6, \Rz:=0), v200, z200, Tooldata_7;
MoveJ RelTool (starting_position, 93, 138.3, -595 \Rx:=-7.3, \Ry:=-7.2, \Rz:=0), v200, z200, Tooldata_7;
MoveJ RelTool (starting_position, 91, 139.1, -595 \Rx:=-7.2, \Ry:=-7.5, \Rz:=0), v200, z200, Tooldata_7;
MoveJ RelTool (starting_position, 88, 139.8, -594 \Rx:=-7.1, \Ry:=-7.8, \Rz:=0), v200, z200, Tooldata_7;
MoveJ RelTool (starting_position, 86, 140.5, -594 \Rx:=-7, \Ry:=-8.4, \Rz:=0), v200, z200, Tooldata_7;
MoveJ RelTool (starting_position, 83, 141.1, -594 \Rx:=-6.8, \Ry:=-8.7, \Rz:=0), v200, z200, Tooldata_7;
MoveJ RelTool (starting_position, 80, 141.8, -593 \Rx:=-6.6, \Ry:=-9.3, \Rz:=0), v200, z200, Tooldata_7;
MoveJ RelTool (starting_position, 77, 142.4, -593 \Rx:=-6.5, \Ry:=-9.9, \Rz:=0), v200, z200, Tooldata_7;
MoveJ RelTool (starting_position, 73, 143, -592 \Rx:=-6.3, \Ry:=-10.5, \Rz:=0), v200, z200, Tooldata_7;
MoveJ RelTool (starting_position, 70, 143.6, -592 \Rx:=-6.2, \Ry:=-11.1, \Rz:=0), v200, z200, Tooldata_7;
MoveJ RelTool (starting_position, 66, 144.1, -592 \Rx:=-6.1, \Ry:=-11.7, \Rz:=0), v200, z200, Tooldata_7;
MoveJ RelTool (starting_position, 63, 144.6, -591 \Rx:=-6.1, \Ry:=-12.3, \Rz:=0), v200, z200, Tooldata_7;
MoveJ RelTool (starting_position, 59, 145.1, -590 \Rx:=-6.1, \Ry:=-12.9, \Rz:=0), v200, z200, Tooldata_7;
MoveJ RelTool (starting_position, 56, 145.6, -590 \Rx:=-6.1, \Ry:=-13.5, \Rz:=0), v200, z200, Tooldata_7;
MoveJ RelTool (starting_position, 52, 146, -589 \Rx:=-6.2, \Ry:=-14.1, \Rz:=0), v200, z200, Tooldata_7;
MoveJ RelTool (starting_position, 49, 146.4, -588 \Rx:=-6.4, \Ry:=-14.7, \Rz:=0), v200, z200, Tooldata_7;
MoveJ RelTool (starting_position, 45, 146.8, -586 \Rx:=-6.6, \Ry:=-15.3, \Rz:=0), v200, z200, Tooldata_7;
MoveJ RelTool (starting_position, 41, 147.1, -585 \Rx:=-6.9, \Ry:=-16.2, \Rz:=0), v200, z200, Tooldata_7;
MoveJ RelTool (starting_position, 38, 147.5, -583 \Rx:=-7.2, \Ry:=-16.8, \Rz:=0), v200, z200, Tooldata_7;
MoveJ RelTool (starting_position, 34, 147.7, -581 \Rx:=-7.5, \Ry:=-17.4, \Rz:=0), v200, z200, Tooldata_7;
MoveJ RelTool (starting_position, 32, 148, -579 \Rx:=-7.9, \Ry:=-17.7, \Rz:=0), v200, z200, Tooldata_7;
MoveJ RelTool (starting_position, 29, 148.3, -577 \Rx:=-8.2, \Ry:=-18.3, \Rz:=0), v200, z200, Tooldata_7;
MoveJ RelTool (starting_position, 26, 148.5, -574 \Rx:=-8.6, \Ry:=-18.6, \Rz:=0), v200, z200, Tooldata_7;
MoveJ RelTool (starting_position, 24, 148.7, -571 \Rx:=-8.9, \Ry:=-19.2, \Rz:=0), v200, z200, Tooldata_7;
MoveJ RelTool (starting_position, 22, 148.9, -568 \Rx:=-9.2, \Ry:=-19.5, \Rz:=0), v200, z200, Tooldata_7;
MoveJ RelTool (starting_position, 21, 149, -565 \Rx:=-9.5, \Ry:=-19.8, \Rz:=0), v200, z200, Tooldata_7;
MoveJ RelTool (starting_position, 20, 149.2, -561 \Rx:=-9.7, \Ry:=-19.8, \Rz:=0), v200, z200, Tooldata_7;
MoveJ RelTool (starting_position, 19, 149.3, -557 \Rx:=-9.9, \Ry:=-20.1, \Rz:=0), v200, z200, Tooldata_7;
MoveJ RelTool (starting_position, 19, 149.5, -553 \Rx:=-10, \Ry:=-20.1, \Rz:=0), v200, z200, Tooldata_7;
MoveJ RelTool (starting_position, 19, 149.6, -549 \Rx:=-10.1, \Ry:=-20.1, \Rz:=0), v200, z200, Tooldata_7;
MoveJ RelTool (starting_position, 20, 149.8, -545 \Rx:=-10.2, \Ry:=-19.8, \Rz:=0), v200, z200, Tooldata_7;
MoveJ RelTool (starting_position, 21, 149.9, -541 \Rx:=-10.2, \Ry:=-19.5, \Rz:=0), v200, z200, Tooldata_7;
MoveJ RelTool (starting_position, 23, 150, -537 \Rx:=-10.1, \Ry:=-19.2, \Rz:=0), v200, z200, Tooldata_7;
MoveJ RelTool (starting_position, 25, 150.2, -533 \Rx:=-10, \Ry:=-18.9, \Rz:=0), v200, z200, Tooldata_7;
MoveJ RelTool (starting_position, 28, 150.3, -529 \Rx:=-9.9, \Ry:=-18.6, \Rz:=0), v200, z200, Tooldata_7;
MoveJ RelTool (starting_position, 30, 150.5, -526 \Rx:=-9.7, \Ry:=-18, \Rz:=0), v200, z200, Tooldata_7;
MoveJ RelTool (starting_position, 34, 150.6, -522 \Rx:=-9.5, \Ry:=-17.4, \Rz:=0), v200, z200, Tooldata_7;
MoveJ RelTool (starting_position, 38, 150.8, -519 \Rx:=-9.3, \Ry:=-16.8, \Rz:=0), v200, z200, Tooldata_7;
MoveJ RelTool (starting_position, 42, 150.9, -516 \Rx:=-9, \Ry:=-15.9, \Rz:=0), v200, z200, Tooldata_7;
MoveJ RelTool (starting_position, 46, 151.1, -513 \Rx:=-8.8, \Ry:=-15.3, \Rz:=0), v200, z200, Tooldata_7;
MoveJ RelTool (starting_position, 51, 151.3, -511 \Rx:=-8.6, \Ry:=-14.4, \Rz:=0), v200, z200, Tooldata_7;
MoveJ RelTool (starting_position, 56, 151.5, -508 \Rx:=-8.4, \Ry:=-13.5, \Rz:=0), v200, z200, Tooldata_7;
MoveJ RelTool (starting_position, 61, 151.7, -506 \Rx:=-8.2, \Ry:=-12.6, \Rz:=0), v200, z200, Tooldata_7;
MoveJ RelTool (starting_position, 66, 151.9, -505 \Rx:=-8, \Ry:=-11.7, \Rz:=0), v200, z200, Tooldata_7;
MoveJ RelTool (starting_position, 71, 152.2, -504 \Rx:=-7.8, \Ry:=-10.8, \Rz:=0), v200, z200, Tooldata_7;
MoveJ RelTool (starting_position, 76, 152.5, -503 \Rx:=-7.7, \Ry:=-9.9, \Rz:=0), v200, z200, Tooldata_7;
MoveJ RelTool (starting_position, 81, 152.8, -502 \Rx:=-7.7, \Ry:=-9, \Rz:=0), v200, z200, Tooldata_7;
MoveJ RelTool (starting_position, 86, 153.2, -501 \Rx:=-7.6, \Ry:=-8.1, \Rz:=0), v200, z200, Tooldata_7;
MoveJ RelTool (starting_position, 90, 153.6, -501 \Rx:=-7.5, \Ry:=-7.5, \Rz:=0), v200, z200, Tooldata_7;
MoveJ RelTool (starting_position, 95, 154, -501 \Rx:=-7.4, \Ry:=-6.6, \Rz:=0), v200, z200, Tooldata_7;
MoveJ RelTool (starting_position, 98, 154.4, -502 \Rx:=-7.4, \Ry:=-6, \Rz:=0), v200, z200, Tooldata_7;
MoveJ RelTool (starting_position, 102, 154.8, -502 \Rx:=-7.4, \Ry:=-5.4, \Rz:=0), v200, z200, Tooldata_7;
MoveJ RelTool (starting_position, 105, 155.3, -503 \Rx:=-7.4, \Ry:=-4.8, \Rz:=0), v200, z200, Tooldata_7;
MoveJ RelTool (starting_position, 108, 155.9, -504 \Rx:=-7.4, \Ry:=-4.2, \Rz:=0), v200, z200, Tooldata_7;
MoveJ RelTool (starting_position, 111, 156.4, -505 \Rx:=-7.4, \Ry:=-3.9, \Rz:=0), v200, z200, Tooldata_7;
MoveJ RelTool (starting_position, 113, 157, -505 \Rx:=-7.4, \Ry:=-3.6, \Rz:=0), v200, z200, Tooldata_7;
MoveJ RelTool (starting_position, 115, 157.6, -506 \Rx:=-7.4, \Ry:=-3, \Rz:=0), v200, z200, Tooldata_7;
MoveJ RelTool (starting_position, 116, 158.2, -507 \Rx:=-7.4, \Ry:=-2.7, \Rz:=0), v200, z200, Tooldata_7;
MoveJ RelTool (starting_position, 117, 158.8, -508 \Rx:=-7.3, \Ry:=-2.7, \Rz:=0), v200, z200, Tooldata_7;
MoveJ RelTool (starting_position, 118, 159.5, -509 \Rx:=-7.2, \Ry:=-2.7, \Rz:=0), v200, z200, Tooldata_7;
MoveJ RelTool (starting_position, 118, 160.2, -510 \Rx:=-7.1, \Ry:=-2.7, \Rz:=0), v200, z200, Tooldata_7;
MoveJ RelTool (starting_position, 118, 160.9, -511 \Rx:=-7, \Ry:=-2.7, \Rz:=0), v200, z200, Tooldata_7;
MoveJ RelTool (starting_position, 118, 161.6, -511 \Rx:=-6.8, \Ry:=-2.7, \Rz:=0), v200, z200, Tooldata_7;
MoveJ RelTool (starting_position, 118, 162.4, -512 \Rx:=-6.6, \Ry:=-2.7, \Rz:=0), v200, z200, Tooldata_7;
MoveJ RelTool (starting_position, 117, 163.1, -512 \Rx:=-6.4, \Ry:=-2.7, \Rz:=0), v200, z200, Tooldata_7;
MoveJ RelTool (starting_position, 117, 163.8, -512 \Rx:=-6.1, \Ry:=-3, \Rz:=0), v200, z200, Tooldata_7;
MoveJ RelTool (starting_position, 116, 164.6, -512 \Rx:=-5.8, \Ry:=-3, \Rz:=0), v200, z200, Tooldata_7;
MoveJ RelTool (starting_position, 115, 165.4, -511 \Rx:=-5.5, \Ry:=-3.3, \Rz:=0), v200, z200, Tooldata_7;
MoveJ RelTool (starting_position, 114, 166.1, -511 \Rx:=-5.2, \Ry:=-3.3, \Rz:=0), v200, z200, Tooldata_7;
MoveJ RelTool (starting_position, 113, 166.9, -510 \Rx:=-4.8, \Ry:=-3.6, \Rz:=0), v200, z200, Tooldata_7;
MoveJ RelTool (starting_position, 112, 167.6, -509 \Rx:=-4.4, \Ry:=-3.9, \Rz:=0), v200, z200, Tooldata_7;
MoveJ RelTool (starting_position, 111, 168.3, -508 \Rx:=-4, \Ry:=-3.9, \Rz:=0), v200, z200, Tooldata_7;
MoveJ RelTool (starting_position, 110, 169.1, -507 \Rx:=-3.7, \Ry:=-4.2, \Rz:=0), v200, z200, Tooldata_7;
MoveJ RelTool (starting_position, 109, 169.8, -505 \Rx:=-3.4, \Ry:=-4.5, \Rz:=0), v200, z200, Tooldata_7;
MoveJ RelTool (starting_position, 108, 170.5, -504 \Rx:=-3.1, \Ry:=-4.5, \Rz:=0), v200, z200, Tooldata_7;
MoveJ RelTool (starting_position, 107, 171.1, -502 \Rx:=-2.9, \Ry:=-4.8, \Rz:=0), v200, z200, Tooldata_7;
MoveJ RelTool (starting_position, 106, 171.8, -501 \Rx:=-2.7, \Ry:=-4.8, \Rz:=0), v200, z200, Tooldata_7;
MoveJ RelTool (starting_position, 106, 172.4, -500 \Rx:=-2.5, \Ry:=-4.8, \Rz:=0), v200, z200, Tooldata_7;
MoveJ RelTool (starting_position, 106, 173, -498 \Rx:=-2.3, \Ry:=-4.8, \Rz:=0), v200, z200, Tooldata_7;
MoveJ RelTool (starting_position, 105, 173.6, -497 \Rx:=-2.1, \Ry:=-5.1, \Rz:=0), v200, z200, Tooldata_7;
MoveJ RelTool (starting_position, 106, 174.1, -496 \Rx:=-2, \Ry:=-5.1, \Rz:=0), v200, z200, Tooldata_7;
MoveJ RelTool (starting_position, 106, 174.6, -494 \Rx:=-1.8, \Ry:=-4.8, \Rz:=0), v200, z200, Tooldata_7;
MoveJ RelTool (starting_position, 107, 175.1, -493 \Rx:=-1.7, \Ry:=-4.8, \Rz:=0), v200, z200, Tooldata_7;
MoveJ RelTool (starting_position, 107, 175.6, -492 \Rx:=-1.6, \Ry:=-4.5, \Rz:=0), v200, z200, Tooldata_7;
MoveJ RelTool (starting_position, 108, 176, -491 \Rx:=-1.4, \Ry:=-4.5, \Rz:=0), v200, z200, Tooldata_7;
MoveJ RelTool (starting_position, 110, 176.4, -491 \Rx:=-1.4, \Ry:=-4.2, \Rz:=0), v200, z200, Tooldata_7;
MoveJ RelTool (starting_position, 111, 176.8, -490 \Rx:=-1.4, \Ry:=-3.9, \Rz:=0), v200, z200, Tooldata_7;
MoveJ RelTool (starting_position, 112, 177.1, -489 \Rx:=-1.4, \Ry:=-3.9, \Rz:=0), v200, z200, Tooldata_7;
MoveJ RelTool (starting_position, 113, 177.5, -489 \Rx:=-1.4, \Ry:=-3.6, \Rz:=0), v200, z200, Tooldata_7;
MoveJ RelTool (starting_position, 115, 177.7, -489 \Rx:=-1.4, \Ry:=-3.3, \Rz:=0), v200, z200, Tooldata_7;
MoveJ RelTool (starting_position, 116, 178, -489 \Rx:=-1.5, \Ry:=-3, \Rz:=0), v200, z200, Tooldata_7;
MoveJ RelTool (starting_position, 118, 178.3, -488 \Rx:=-1.5, \Ry:=-2.7, \Rz:=0), v200, z200, Tooldata_7;
MoveJ RelTool (starting_position, 120, 178.5, -488 \Rx:=-1.6, \Ry:=-2.4, \Rz:=0), v200, z200, Tooldata_7;
MoveJ RelTool (starting_position, 121, 178.7, -488 \Rx:=-1.6, \Ry:=-2.1, \Rz:=0), v200, z200, Tooldata_7;
MoveJ RelTool (starting_position, 123, 178.9, -488 \Rx:=-1.8, \Ry:=-2.1, \Rz:=0), v200, z200, Tooldata_7;
MoveJ RelTool (starting_position, 124, 179, -489 \Rx:=-1.8, \Ry:=-1.5, \Rz:=0), v200, z200, Tooldata_7;
MoveJ RelTool (starting_position, 125, 179.2, -489 \Rx:=-1.9, \Ry:=-1.5, \Rz:=0), v200, z200, Tooldata_7;
MoveJ RelTool (starting_position, 127, 179.3, -489 \Rx:=-2.1, \Ry:=-1.2, \Rz:=0), v200, z200, Tooldata_7;
MoveJ RelTool (starting_position, 128, 179.4, -489 \Rx:=-2.2, \Ry:=-0.9, \Rz:=0), v200, z200, Tooldata_7;
MoveJ RelTool (starting_position, 130, 179.5, -489 \Rx:=-2.4, \Ry:=-0.6, \Rz:=0), v200, z200, Tooldata_7;
MoveJ RelTool (starting_position, 131, 179.6, -489 \Rx:=-2.6, \Ry:=-0.3, \Rz:=0), v200, z200, Tooldata_7;
MoveJ RelTool (starting_position, 132, 179.7, -490 \Rx:=-2.8, \Ry:=-0.3, \Rz:=0), v200, z200, Tooldata_7;
MoveJ RelTool (starting_position, 134, 179.8, -490 \Rx:=-3, \Ry:=-0, \Rz:=0), v200, z200, Tooldata_7;
MoveJ RelTool (starting_position, 135, 179.9, -490 \Rx:=-3.3, \Ry:=0.3, \Rz:=0), v200, z200, Tooldata_7;
MoveJ RelTool (starting_position, 136, 180, -490 \Rx:=-3.6, \Ry:=0.3, \Rz:=0), v200, z200, Tooldata_7;
MoveJ RelTool (starting_position, 138, 180.1, -490 \Rx:=-3.9, \Ry:=0.6, \Rz:=0), v200, z200, Tooldata_7;
MoveJ RelTool (starting_position, 139, 180.2, -490 \Rx:=-4.3, \Ry:=0.9, \Rz:=0), v200, z200, Tooldata_7;
MoveJ RelTool (starting_position, 141, 180.3, -490 \Rx:=-4.7, \Ry:=1.2, \Rz:=0), v200, z200, Tooldata_7;
MoveJ RelTool (starting_position, 142, 180.3, -490 \Rx:=-5.2, \Ry:=1.5, \Rz:=0), v200, z200, Tooldata_7;
MoveJ RelTool (starting_position, 144, 180.4, -490 \Rx:=-5.7, \Ry:=1.8, \Rz:=0), v200, z200, Tooldata_7;
MoveJ RelTool (starting_position, 146, 180.5, -490 \Rx:=-6.2, \Ry:=2.1, \Rz:=0), v200, z200, Tooldata_7;
MoveJ RelTool (starting_position, 147, 180.7, -490 \Rx:=-6.7, \Ry:=2.4, \Rz:=0), v200, z200, Tooldata_7;
MoveJ RelTool (starting_position, 149, 180.8, -490 \Rx:=-7.3, \Ry:=2.7, \Rz:=0), v200, z200, Tooldata_7;
MoveJ RelTool (starting_position, 150, 180.9, -490 \Rx:=-7.9, \Ry:=3, \Rz:=0), v200, z200, Tooldata_7;
MoveJ RelTool (starting_position, 152, 181.1, -490 \Rx:=-8.4, \Ry:=3, \Rz:=0), v200, z200, Tooldata_7;
MoveJ RelTool (starting_position, 153, 181.3, -490 \Rx:=-9, \Ry:=3.3, \Rz:=0), v200, z200, Tooldata_7;
MoveJ RelTool (starting_position, 155, 181.5, -491 \Rx:=-9.6, \Ry:=3.6, \Rz:=0), v200, z200, Tooldata_7;
MoveJ RelTool (starting_position, 156, 181.7, -491 \Rx:=-10.2, \Ry:=3.9, \Rz:=0), v200, z200, Tooldata_7;
MoveJ RelTool (starting_position, 158, 181.9, -491 \Rx:=-10.8, \Ry:=4.2, \Rz:=0), v200, z200, Tooldata_7;
MoveJ RelTool (starting_position, 159, 182.2, -491 \Rx:=-11.4, \Ry:=4.5, \Rz:=0), v200, z200, Tooldata_7;
MoveJ RelTool (starting_position, 161, 182.5, -492 \Rx:=-11.9, \Ry:=4.8, \Rz:=0), v200, z200, Tooldata_7;
MoveJ RelTool (starting_position, 162, 182.8, -492 \Rx:=-12.3, \Ry:=4.8, \Rz:=0), v200, z200, Tooldata_7;
MoveJ RelTool (starting_position, 163, 183.2, -493 \Rx:=-12.7, \Ry:=5.1, \Rz:=0), v200, z200, Tooldata_7;
MoveJ RelTool (starting_position, 165, 183.6, -493 \Rx:=-12.9, \Ry:=5.4, \Rz:=0), v200, z200, Tooldata_7;
MoveJ RelTool (starting_position, 166, 184, -494 \Rx:=-13.2, \Ry:=5.7, \Rz:=0), v200, z200, Tooldata_7;
MoveJ RelTool (starting_position, 168, 184.4, -495 \Rx:=-13.4, \Ry:=6, \Rz:=0), v200, z200, Tooldata_7;
MoveJ RelTool (starting_position, 169, 184.8, -495 \Rx:=-13.5, \Ry:=6, \Rz:=0), v200, z200, Tooldata_7;
MoveJ RelTool (starting_position, 170, 185.3, -496 \Rx:=-13.5, \Ry:=6.3, \Rz:=0), v200, z200, Tooldata_7;
MoveJ RelTool (starting_position, 171, 185.9, -497 \Rx:=-13.5, \Ry:=6.6, \Rz:=0), v200, z200, Tooldata_7;
MoveJ RelTool (starting_position, 172, 186.4, -498 \Rx:=-13.4, \Ry:=6.6, \Rz:=0), v200, z200, Tooldata_7;
MoveJ RelTool (starting_position, 173, 187, -499 \Rx:=-13.2, \Ry:=6.9, \Rz:=0), v200, z200, Tooldata_7;
MoveJ RelTool (starting_position, 174, 187.6, -500 \Rx:=-13, \Ry:=6.9, \Rz:=0), v200, z200, Tooldata_7;
MoveJ RelTool (starting_position, 175, 188.2, -501 \Rx:=-12.7, \Ry:=7.2, \Rz:=0), v200, z200, Tooldata_7;
MoveJ RelTool (starting_position, 176, 188.8, -502 \Rx:=-12.4, \Ry:=7.2, \Rz:=0), v200, z200, Tooldata_7;
MoveJ RelTool (starting_position, 176, 189.5, -503 \Rx:=-11.9, \Ry:=7.5, \Rz:=0), v200, z200, Tooldata_7;
MoveJ RelTool (starting_position, 177, 190.2, -504 \Rx:=-11.3, \Ry:=7.5, \Rz:=0), v200, z200, Tooldata_7;
MoveJ RelTool (starting_position, 177, 190.9, -505 \Rx:=-10.7, \Ry:=7.5, \Rz:=0), v200, z200, Tooldata_7;
MoveJ RelTool (starting_position, 177, 191.6, -506 \Rx:=-10.1, \Ry:=7.5, \Rz:=0), v200, z200, Tooldata_7;
MoveJ RelTool (starting_position, 177, 192.4, -507 \Rx:=-9.5, \Ry:=7.5, \Rz:=0), v200, z200, Tooldata_7;
MoveJ RelTool (starting_position, 177, 193.1, -508 \Rx:=-8.8, \Ry:=7.5, \Rz:=0), v200, z200, Tooldata_7;
MoveJ RelTool (starting_position, 177, 193.8, -509 \Rx:=-8, \Ry:=7.5, \Rz:=0), v200, z200, Tooldata_7;
MoveJ RelTool (starting_position, 177, 194.6, -510 \Rx:=-7.3, \Ry:=7.5, \Rz:=0), v200, z200, Tooldata_7;
MoveJ RelTool (starting_position, 177, 195.4, -512 \Rx:=-6.5, \Ry:=7.5, \Rz:=0), v200, z200, Tooldata_7;
MoveJ RelTool (starting_position, 177, 196.1, -513 \Rx:=-5.6, \Ry:=7.5, \Rz:=0), v200, z200, Tooldata_7;
MoveJ RelTool (starting_position, 176, 196.9, -514 \Rx:=-4.8, \Ry:=7.5, \Rz:=0), v200, z200, Tooldata_7;
MoveJ RelTool (starting_position, 175, 197.6, -515 \Rx:=-3.9, \Ry:=7.2, \Rz:=0), v200, z200, Tooldata_7;
MoveJ RelTool (starting_position, 175, 198.3, -516 \Rx:=-3, \Ry:=7.2, \Rz:=0), v200, z200, Tooldata_7;
MoveJ RelTool (starting_position, 174, 199.1, -517 \Rx:=-2.1, \Ry:=6.9, \Rz:=0), v200, z200, Tooldata_7;
MoveJ RelTool (starting_position, 172, 199.8, -518 \Rx:=-1.3, \Ry:=6.6, \Rz:=0), v200, z200, Tooldata_7;
MoveJ RelTool (starting_position, 171, 200.5, -519 \Rx:=-0.5, \Ry:=6.6, \Rz:=0), v200, z200, Tooldata_7;
MoveJ RelTool (starting_position, 170, 201.1, -520 \Rx:=0.3, \Ry:=6.3, \Rz:=0), v200, z200, Tooldata_7;
MoveJ RelTool (starting_position, 168, 201.8, -521 \Rx:=1.1, \Ry:=6, \Rz:=0), v200, z200, Tooldata_7;
MoveJ RelTool (starting_position, 167, 202.4, -522 \Rx:=1.8, \Ry:=5.7, \Rz:=0), v200, z200, Tooldata_7;
MoveJ RelTool (starting_position, 165, 203, -523 \Rx:=2.5, \Ry:=5.4, \Rz:=0), v200, z200, Tooldata_7;
MoveJ RelTool (starting_position, 164, 203.6, -523 \Rx:=3.1, \Ry:=5.4, \Rz:=0), v200, z200, Tooldata_7;
MoveJ RelTool (starting_position, 162, 204.1, -524 \Rx:=3.7, \Ry:=5.1, \Rz:=0), v200, z200, Tooldata_7;
MoveJ RelTool (starting_position, 161, 204.6, -524 \Rx:=4.1, \Ry:=4.5, \Rz:=0), v200, z200, Tooldata_7;
MoveJ RelTool (starting_position, 159, 205.1, -525 \Rx:=4.6, \Ry:=4.2, \Rz:=0), v200, z200, Tooldata_7;
MoveJ RelTool (starting_position, 158, 205.6, -525 \Rx:=5, \Ry:=4.2, \Rz:=0), v200, z200, Tooldata_7;
MoveJ RelTool (starting_position, 157, 206, -525 \Rx:=5.4, \Ry:=3.9, \Rz:=0), v200, z200, Tooldata_7;
MoveJ RelTool (starting_position, 156, 206.4, -525 \Rx:=5.6, \Ry:=3.9, \Rz:=0), v200, z200, Tooldata_7;
MoveJ RelTool (starting_position, 154, 206.8, -526 \Rx:=5.8, \Ry:=3.6, \Rz:=0), v200, z200, Tooldata_7;
MoveJ RelTool (starting_position, 153, 207.1, -526 \Rx:=6, \Ry:=3.3, \Rz:=0), v200, z200, Tooldata_7;
MoveJ RelTool (starting_position, 152, 207.5, -526 \Rx:=6, \Ry:=3, \Rz:=0), v200, z200, Tooldata_7;
MoveJ RelTool (starting_position, 151, 207.7, -526 \Rx:=5.9, \Ry:=3, \Rz:=0), v200, z200, Tooldata_7;
MoveJ RelTool (starting_position, 150, 208, -526 \Rx:=5.9, \Ry:=2.7, \Rz:=0), v200, z200, Tooldata_7;
MoveJ RelTool (starting_position, 150, 208.3, -526 \Rx:=5.7, \Ry:=2.7, \Rz:=0), v200, z200, Tooldata_7;
MoveJ RelTool (starting_position, 149, 208.5, -526 \Rx:=5.5, \Ry:=2.7, \Rz:=0), v200, z200, Tooldata_7;
MoveJ RelTool (starting_position, 149, 208.7, -525 \Rx:=5.2, \Ry:=2.7, \Rz:=0), v200, z200, Tooldata_7;
MoveJ RelTool (starting_position, 148, 208.9, -525 \Rx:=5, \Ry:=2.4, \Rz:=0), v200, z200, Tooldata_7;
MoveJ RelTool (starting_position, 148, 209, -525 \Rx:=4.8, \Ry:=2.4, \Rz:=0), v200, z200, Tooldata_7;
MoveJ RelTool (starting_position, 148, 209.2, -525 \Rx:=4.5, \Ry:=2.4, \Rz:=0), v200, z200, Tooldata_7;
MoveJ RelTool (starting_position, 148, 209.3, -526 \Rx:=4.3, \Ry:=2.4, \Rz:=0), v200, z200, Tooldata_7;
MoveJ RelTool (starting_position, 149, 209.4, -526 \Rx:=4.1, \Ry:=2.7, \Rz:=0), v200, z200, Tooldata_7;
MoveJ RelTool (starting_position, 149, 209.5, -526 \Rx:=3.9, \Ry:=2.7, \Rz:=0), v200, z200, Tooldata_7;
MoveJ RelTool (starting_position, 149, 209.6, -526 \Rx:=3.7, \Ry:=2.7, \Rz:=0), v200, z200, Tooldata_7;
MoveJ RelTool (starting_position, 150, 209.7, -526 \Rx:=3.6, \Ry:=2.7, \Rz:=0), v200, z200, Tooldata_7;
MoveJ RelTool (starting_position, 150, 209.8, -526 \Rx:=3.6, \Ry:=2.7, \Rz:=0), v200, z200, Tooldata_7;
MoveJ RelTool (starting_position, 150, 209.8, -527 \Rx:=3.6, \Ry:=3, \Rz:=0), v200, z200, Tooldata_7;
MoveJ RelTool (starting_position, 151, 209.9, -527 \Rx:=3.7, \Ry:=3, \Rz:=0), v200, z200, Tooldata_7;
MoveJ RelTool (starting_position, 151, 209.9, -527 \Rx:=3.8, \Ry:=3, \Rz:=0), v200, z200, Tooldata_7;
MoveJ RelTool (starting_position, 152, 210, -528 \Rx:=3.9, \Ry:=3, \Rz:=0), v200, z200, Tooldata_7;
MoveJ RelTool (starting_position, 152, 210, -528 \Rx:=4, \Ry:=3.3, \Rz:=0), v200, z200, Tooldata_7;
MoveJ RelTool (starting_position, 153, 210, -529 \Rx:=4.2, \Ry:=3.3, \Rz:=0), v200, z200, Tooldata_7;
MoveJ RelTool (starting_position, 153, 210, -529 \Rx:=4.4, \Ry:=3.3, \Rz:=0), v200, z200, Tooldata_7;
MoveJ RelTool (starting_position, 153, 210, -530 \Rx:=4.6, \Ry:=3.3, \Rz:=0), v200, z200, Tooldata_7;
MoveJ RelTool (starting_position, 154, 210, -531 \Rx:=4.8, \Ry:=3.6, \Rz:=0), v200, z200, Tooldata_7;
MoveJ RelTool (starting_position, 154, 210, -531 \Rx:=4.9, \Ry:=3.6, \Rz:=0), v200, z200, Tooldata_7;
MoveJ RelTool (starting_position, 154, 210.1, -532 \Rx:=5, \Ry:=3.6, \Rz:=0), v200, z200, Tooldata_7;
MoveJ RelTool (starting_position, 154, 210.1, -532 \Rx:=5.1, \Ry:=3.6, \Rz:=0), v200, z200, Tooldata_7;
MoveJ RelTool (starting_position, 155, 210.2, -533 \Rx:=5.2, \Ry:=3.6, \Rz:=0), v200, z200, Tooldata_7;
MoveJ RelTool (starting_position, 155, 210.3, -534 \Rx:=5.2, \Ry:=3.6, \Rz:=0), v200, z200, Tooldata_7;
MoveJ RelTool (starting_position, 154, 210.3, -534 \Rx:=5.2, \Ry:=3.6, \Rz:=0), v200, z200, Tooldata_7;
MoveJ RelTool (starting_position, 154, 210.4, -535 \Rx:=5.2, \Ry:=3.6, \Rz:=0), v200, z200, Tooldata_7;
MoveJ RelTool (starting_position, 154, 210.5, -535 \Rx:=5.2, \Ry:=3.6, \Rz:=0), v200, z200, Tooldata_7;
MoveJ RelTool (starting_position, 154, 210.7, -536 \Rx:=5.2, \Ry:=3.6, \Rz:=0), v200, z200, Tooldata_7;
MoveJ RelTool (starting_position, 153, 210.8, -537 \Rx:=5.3, \Ry:=3.3, \Rz:=0), v200, z200, Tooldata_7;
MoveJ RelTool (starting_position, 153, 210.9, -537 \Rx:=5.3, \Ry:=3.3, \Rz:=0), v200, z200, Tooldata_7;
MoveJ RelTool (starting_position, 153, 211.1, -538 \Rx:=5.3, \Ry:=3.3, \Rz:=0), v200, z200, Tooldata_7;
MoveJ RelTool (starting_position, 152, 211.3, -539 \Rx:=5.4, \Ry:=3.3, \Rz:=0), v200, z200, Tooldata_7;
MoveJ RelTool (starting_position, 152, 211.5, -539 \Rx:=5.5, \Ry:=3, \Rz:=0), v200, z200, Tooldata_7;
MoveJ RelTool (starting_position, 151, 211.7, -540 \Rx:=5.6, \Ry:=3, \Rz:=0), v200, z200, Tooldata_7;
MoveJ RelTool (starting_position, 150, 211.9, -540 \Rx:=5.8, \Ry:=3, \Rz:=0), v200, z200, Tooldata_7;
MoveJ RelTool (starting_position, 149, 212.2, -541 \Rx:=6.1, \Ry:=2.7, \Rz:=0), v200, z200, Tooldata_7;
MoveJ RelTool (starting_position, 148, 212.5, -542 \Rx:=6.3, \Ry:=2.4, \Rz:=0), v200, z200, Tooldata_7;
MoveJ RelTool (starting_position, 147, 212.8, -542 \Rx:=6.6, \Ry:=2.1, \Rz:=0), v200, z200, Tooldata_7;
MoveJ RelTool (starting_position, 146, 213.2, -542 \Rx:=6.9, \Ry:=2.1, \Rz:=0), v200, z200, Tooldata_7;
MoveJ RelTool (starting_position, 144, 213.6, -543 \Rx:=7.2, \Ry:=1.8, \Rz:=0), v200, z200, Tooldata_7;
MoveJ RelTool (starting_position, 143, 214, -543 \Rx:=7.5, \Ry:=1.8, \Rz:=0), v200, z200, Tooldata_7;
MoveJ RelTool (starting_position, 142, 214.4, -544 \Rx:=7.8, \Ry:=1.5, \Rz:=0), v200, z200, Tooldata_7;
MoveJ RelTool (starting_position, 140, 214.8, -544 \Rx:=8, \Ry:=1.2, \Rz:=0), v200, z200, Tooldata_7;
MoveJ RelTool (starting_position, 139, 215.3, -544 \Rx:=8.3, \Ry:=0.6, \Rz:=0), v200, z200, Tooldata_7;
MoveJ RelTool (starting_position, 137, 215.9, -544 \Rx:=8.6, \Ry:=0.6, \Rz:=0), v200, z200, Tooldata_7;
MoveJ RelTool (starting_position, 135, 216.4, -544 \Rx:=8.8, \Ry:=0.3, \Rz:=0), v200, z200, Tooldata_7;
MoveJ RelTool (starting_position, 134, 217, -544 \Rx:=8.9, \Ry:=-0, \Rz:=0), v200, z200, Tooldata_7;
MoveJ RelTool (starting_position, 132, 217.6, -544 \Rx:=9, \Ry:=-0.3, \Rz:=0), v200, z200, Tooldata_7;
MoveJ RelTool (starting_position, 130, 218.2, -544 \Rx:=9, \Ry:=-0.6, \Rz:=0), v200, z200, Tooldata_7;
MoveJ RelTool (starting_position, 128, 218.8, -544 \Rx:=9, \Ry:=-1.2, \Rz:=0), v200, z200, Tooldata_7;
MoveJ RelTool (starting_position, 127, 219.5, -544 \Rx:=8.9, \Ry:=-1.2, \Rz:=0), v200, z200, Tooldata_7;
MoveJ RelTool (starting_position, 125, 220.2, -544 \Rx:=8.7, \Ry:=-1.5, \Rz:=0), v200, z200, Tooldata_7;
MoveJ RelTool (starting_position, 123, 220.9, -544 \Rx:=8.5, \Ry:=-1.8, \Rz:=0), v200, z200, Tooldata_7;
MoveJ RelTool (starting_position, 122, 221.6, -543 \Rx:=8.1, \Ry:=-2.1, \Rz:=0), v200, z200, Tooldata_7;
MoveJ RelTool (starting_position, 120, 222.4, -543 \Rx:=7.7, \Ry:=-2.4, \Rz:=0), v200, z200, Tooldata_7;
MoveJ RelTool (starting_position, 118, 223.1, -543 \Rx:=7.4, \Ry:=-2.7, \Rz:=0), v200, z200, Tooldata_7;
MoveJ RelTool (starting_position, 117, 223.8, -542 \Rx:=6.9, \Ry:=-3, \Rz:=0), v200, z200, Tooldata_7;
MoveJ RelTool (starting_position, 115, 224.6, -542 \Rx:=6.4, \Ry:=-3.3, \Rz:=0), v200, z200, Tooldata_7;
MoveJ RelTool (starting_position, 114, 225.4, -542 \Rx:=5.9, \Ry:=-3.3, \Rz:=0), v200, z200, Tooldata_7;
MoveJ RelTool (starting_position, 113, 226.1, -541 \Rx:=5.4, \Ry:=-3.6, \Rz:=0), v200, z200, Tooldata_7;
MoveJ RelTool (starting_position, 112, 226.9, -541 \Rx:=4.8, \Ry:=-3.9, \Rz:=0), v200, z200, Tooldata_7;
MoveJ RelTool (starting_position, 110, 227.6, -540 \Rx:=4.3, \Ry:=-4.2, \Rz:=0), v200, z200, Tooldata_7;
MoveJ RelTool (starting_position, 109, 228.3, -540 \Rx:=3.7, \Ry:=-4.2, \Rz:=0), v200, z200, Tooldata_7;
MoveJ RelTool (starting_position, 108, 229.1, -539 \Rx:=3.1, \Ry:=-4.5, \Rz:=0), v200, z200, Tooldata_7;
MoveJ RelTool (starting_position, 106, 229.8, -539 \Rx:=2.5, \Ry:=-4.8, \Rz:=0), v200, z200, Tooldata_7;
MoveJ RelTool (starting_position, 105, 230.5, -538 \Rx:=1.9, \Ry:=-5.1, \Rz:=0), v200, z200, Tooldata_7;
MoveJ RelTool (starting_position, 103, 231.1, -538 \Rx:=1.3, \Ry:=-5.4, \Rz:=0), v200, z200, Tooldata_7;
MoveJ RelTool (starting_position, 102, 231.8, -537 \Rx:=0.7, \Ry:=-5.4, \Rz:=0), v200, z200, Tooldata_7;
MoveJ RelTool (starting_position, 101, 232.4, -537 \Rx:=0.2, \Ry:=-5.7, \Rz:=0), v200, z200, Tooldata_7;
MoveJ RelTool (starting_position, 99, 233, -536 \Rx:=-0.2, \Ry:=-6, \Rz:=0), v200, z200, Tooldata_7;
MoveJ RelTool (starting_position, 98, 233.6, -536 \Rx:=-0.6, \Ry:=-6.3, \Rz:=0), v200, z200, Tooldata_7;
MoveJ RelTool (starting_position, 97, 234.1, -535 \Rx:=-0.9, \Ry:=-6.6, \Rz:=0), v200, z200, Tooldata_7;
MoveJ RelTool (starting_position, 96, 234.6, -534 \Rx:=-1.2, \Ry:=-6.6, \Rz:=0), v200, z200, Tooldata_7;
MoveJ RelTool (starting_position, 95, 235.1, -534 \Rx:=-1.4, \Ry:=-6.9, \Rz:=0), v200, z200, Tooldata_7;
MoveJ RelTool (starting_position, 94, 235.6, -533 \Rx:=-1.5, \Ry:=-6.9, \Rz:=0), v200, z200, Tooldata_7;
MoveJ RelTool (starting_position, 93, 236, -533 \Rx:=-1.6, \Ry:=-6.9, \Rz:=0), v200, z200, Tooldata_7;
MoveJ RelTool (starting_position, 92, 236.4, -532 \Rx:=-1.7, \Ry:=-7.2, \Rz:=0), v200, z200, Tooldata_7;
MoveJ RelTool (starting_position, 91, 236.8, -531 \Rx:=-1.7, \Ry:=-7.5, \Rz:=0), v200, z200, Tooldata_7;
MoveJ RelTool (starting_position, 90, 237.1, -530 \Rx:=-1.7, \Ry:=-7.5, \Rz:=0), v200, z200, Tooldata_7;
MoveJ RelTool (starting_position, 90, 237.5, -530 \Rx:=-1.6, \Ry:=-7.8, \Rz:=0), v200, z200, Tooldata_7;
MoveJ RelTool (starting_position, 89, 237.7, -529 \Rx:=-1.4, \Ry:=-7.8, \Rz:=0), v200, z200, Tooldata_7;
MoveJ RelTool (starting_position, 89, 238, -528 \Rx:=-1.3, \Ry:=-7.8, \Rz:=0), v200, z200, Tooldata_7;
MoveJ RelTool (starting_position, 89, 238.3, -527 \Rx:=-1.1, \Ry:=-7.8, \Rz:=0), v200, z200, Tooldata_7;
MoveJ RelTool (starting_position, 89, 238.5, -526 \Rx:=-0.9, \Ry:=-7.8, \Rz:=0), v200, z200, Tooldata_7;
MoveJ RelTool (starting_position, 89, 238.7, -525 \Rx:=-0.7, \Ry:=-7.8, \Rz:=0), v200, z200, Tooldata_7;
MoveJ RelTool (starting_position, 89, 238.9, -524 \Rx:=-0.5, \Ry:=-7.8, \Rz:=0), v200, z200, Tooldata_7;
MoveJ RelTool (starting_position, 90, 239, -523 \Rx:=-0.3, \Ry:=-7.5, \Rz:=0), v200, z200, Tooldata_7;
MoveJ RelTool (starting_position, 90, 239.2, -522 \Rx:=-0, \Ry:=-7.5, \Rz:=0), v200, z200, Tooldata_7;
MoveJ RelTool (starting_position, 90, 239.3, -521 \Rx:=0.3, \Ry:=-7.5, \Rz:=0), v200, z200, Tooldata_7;
MoveJ RelTool (starting_position, 90, 239.4, -520 \Rx:=0.6, \Ry:=-7.5, \Rz:=0), v200, z200, Tooldata_7;
MoveJ RelTool (starting_position, 90, 239.5, -519 \Rx:=0.9, \Ry:=-7.5, \Rz:=0), v200, z200, Tooldata_7;
MoveJ RelTool (starting_position, 91, 239.6, -518 \Rx:=1.3, \Ry:=-7.5, \Rz:=0), v200, z200, Tooldata_7;
MoveJ RelTool (starting_position, 91, 239.7, -517 \Rx:=1.6, \Ry:=-7.5, \Rz:=0), v200, z200, Tooldata_7;
MoveJ RelTool (starting_position, 91, 239.8, -516 \Rx:=2, \Ry:=-7.5, \Rz:=0), v200, z200, Tooldata_7;
MoveJ RelTool (starting_position, 91, 239.8, -515 \Rx:=2.4, \Ry:=-7.5, \Rz:=0), v200, z200, Tooldata_7;
MoveJ RelTool (starting_position, 92, 239.9, -514 \Rx:=2.9, \Ry:=-7.2, \Rz:=0), v200, z200, Tooldata_7;
MoveJ RelTool (starting_position, 93, 239.9, -513 \Rx:=3.4, \Ry:=-7.2, \Rz:=0), v200, z200, Tooldata_7;
MoveJ RelTool (starting_position, 94, 240, -512 \Rx:=3.9, \Ry:=-6.9, \Rz:=0), v200, z200, Tooldata_7;
MoveJ RelTool (starting_position, 95, 240, -511 \Rx:=4.4, \Ry:=-6.9, \Rz:=0), v200, z200, Tooldata_7;
MoveJ RelTool (starting_position, 96, 240, -510 \Rx:=4.9, \Ry:=-6.6, \Rz:=0), v200, z200, Tooldata_7;
MoveJ RelTool (starting_position, 97, 240, -509 \Rx:=5.5, \Ry:=-6.3, \Rz:=0), v200, z200, Tooldata_7;
MoveJ RelTool (starting_position, 98, 240, -509 \Rx:=6, \Ry:=-6.3, \Rz:=0), v200, z200, Tooldata_7;
MoveJ RelTool (starting_position, 99, 240, -508 \Rx:=6.6, \Ry:=-6, \Rz:=0), v200, z200, Tooldata_7;
MoveJ RelTool (starting_position, 99, 240, -507 \Rx:=7.2, \Ry:=-6, \Rz:=0), v200, z200, Tooldata_7;
MoveJ RelTool (starting_position, 100, 240, -506 \Rx:=7.8, \Ry:=-5.7, \Rz:=0), v200, z200, Tooldata_7;
MoveJ RelTool (starting_position, 101, 240, -506 \Rx:=8.3, \Ry:=-5.7, \Rz:=0), v200, z200, Tooldata_7;
MoveJ RelTool (starting_position, 102, 240, -505 \Rx:=8.9, \Ry:=-5.4, \Rz:=0), v200, z200, Tooldata_7;
MoveJ RelTool (starting_position, 102, 240, -505 \Rx:=9.4, \Ry:=-5.4, \Rz:=0), v200, z200, Tooldata_7;
MoveJ RelTool (starting_position, 103, 240, -505 \Rx:=10, \Ry:=-5.1, \Rz:=0), v200, z200, Tooldata_7;
MoveJ RelTool (starting_position, 103, 240, -505 \Rx:=10.5, \Ry:=-5.4, \Rz:=0), v200, z200, Tooldata_7;
MoveJ RelTool (starting_position, 103, 240, -504 \Rx:=11, \Ry:=-5.4, \Rz:=0), v200, z200, Tooldata_7;
MoveJ RelTool (starting_position, 103, 240, -504 \Rx:=11.4, \Ry:=-5.4, \Rz:=0), v200, z200, Tooldata_7;
MoveJ RelTool (starting_position, 102, 240, -504 \Rx:=11.9, \Ry:=-5.4, \Rz:=0), v200, z200, Tooldata_7;
MoveJ RelTool (starting_position, 102, 240, -505 \Rx:=12.3, \Ry:=-5.4, \Rz:=0), v200, z200, Tooldata_7;
MoveJ RelTool (starting_position, 101, 240, -505 \Rx:=12.8, \Ry:=-5.7, \Rz:=0), v200, z200, Tooldata_7;
MoveJ RelTool (starting_position, 100, 240, -505 \Rx:=13.1, \Ry:=-5.7, \Rz:=0), v200, z200, Tooldata_7;
MoveJ RelTool (starting_position, 99, 240, -505 \Rx:=13.5, \Ry:=-6, \Rz:=0), v200, z200, Tooldata_7;
MoveJ RelTool (starting_position, 97, 240, -505 \Rx:=13.8, \Ry:=-6.3, \Rz:=0), v200, z200, Tooldata_7;
MoveJ RelTool (starting_position, 95, 240, -506 \Rx:=14.1, \Ry:=-6.6, \Rz:=0), v200, z200, Tooldata_7;
MoveJ RelTool (starting_position, 93, 240, -506 \Rx:=14.3, \Ry:=-6.9, \Rz:=0), v200, z200, Tooldata_7;
MoveJ RelTool (starting_position, 91, 240, -506 \Rx:=14.5, \Ry:=-7.5, \Rz:=0), v200, z200, Tooldata_7;
MoveJ RelTool (starting_position, 89, 240.1, -506 \Rx:=14.7, \Ry:=-7.8, \Rz:=0), v200, z200, Tooldata_7;
MoveJ RelTool (starting_position, 86, 240.1, -505 \Rx:=14.8, \Ry:=-8.1, \Rz:=0), v200, z200, Tooldata_7;
MoveJ RelTool (starting_position, 84, 240.2, -505 \Rx:=14.9, \Ry:=-8.7, \Rz:=0), v200, z200, Tooldata_7;
MoveJ RelTool (starting_position, 81, 240.3, -505 \Rx:=15.1, \Ry:=-9, \Rz:=0), v200, z200, Tooldata_7;
MoveJ RelTool (starting_position, 78, 240.3, -504 \Rx:=15.2, \Ry:=-9.6, \Rz:=0), v200, z200, Tooldata_7;
MoveJ RelTool (starting_position, 75, 240.4, -503 \Rx:=15.3, \Ry:=-10.2, \Rz:=0), v200, z200, Tooldata_7;
MoveJ RelTool (starting_position, 72, 240.5, -502 \Rx:=15.3, \Ry:=-10.8, \Rz:=0), v200, z200, Tooldata_7;
MoveJ RelTool (starting_position, 69, 240.7, -500 \Rx:=15.3, \Ry:=-11.4, \Rz:=0), v200, z200, Tooldata_7;
MoveJ RelTool (starting_position, 66, 240.8, -499 \Rx:=15.3, \Ry:=-11.7, \Rz:=0), v200, z200, Tooldata_7;
MoveJ RelTool (starting_position, 63, 240.9, -497 \Rx:=15.3, \Ry:=-12.3, \Rz:=0), v200, z200, Tooldata_7;
MoveJ RelTool (starting_position, 60, 241.1, -495 \Rx:=15.2, \Ry:=-12.9, \Rz:=0), v200, z200, Tooldata_7;
MoveJ RelTool (starting_position, 57, 241.3, -492 \Rx:=15.1, \Ry:=-13.5, \Rz:=0), v200, z200, Tooldata_7;
MoveJ RelTool (starting_position, 55, 241.5, -490 \Rx:=15, \Ry:=-13.8, \Rz:=0), v200, z200, Tooldata_7;
MoveJ RelTool (starting_position, 53, 241.7, -488 \Rx:=14.8, \Ry:=-14.1, \Rz:=0), v200, z200, Tooldata_7;
MoveJ RelTool (starting_position, 51, 241.9, -485 \Rx:=14.7, \Ry:=-14.4, \Rz:=0), v200, z200, Tooldata_7;
MoveJ RelTool (starting_position, 49, 242.2, -482 \Rx:=14.5, \Ry:=-14.7, \Rz:=0), v200, z200, Tooldata_7;
MoveJ RelTool (starting_position, 48, 242.5, -480 \Rx:=14.2, \Ry:=-15, \Rz:=0), v200, z200, Tooldata_7;
MoveJ RelTool (starting_position, 47, 242.8, -477 \Rx:=14, \Ry:=-15.3, \Rz:=0), v200, z200, Tooldata_7;
MoveJ RelTool (starting_position, 46, 243.2, -474 \Rx:=13.7, \Ry:=-15.3, \Rz:=0), v200, z200, Tooldata_7;
MoveJ RelTool (starting_position, 46, 243.6, -472 \Rx:=13.4, \Ry:=-15.3, \Rz:=0), v200, z200, Tooldata_7;
MoveJ RelTool (starting_position, 46, 244, -469 \Rx:=13.1, \Ry:=-15.3, \Rz:=0), v200, z200, Tooldata_7;
MoveJ RelTool (starting_position, 46, 244.4, -466 \Rx:=12.7, \Ry:=-15.3, \Rz:=0), v200, z200, Tooldata_7;
MoveJ RelTool (starting_position, 46, 244.8, -464 \Rx:=12.3, \Ry:=-15.3, \Rz:=0), v200, z200, Tooldata_7;
MoveJ RelTool (starting_position, 46, 245.3, -461 \Rx:=11.9, \Ry:=-15.3, \Rz:=0), v200, z200, Tooldata_7;
MoveJ RelTool (starting_position, 47, 245.9, -459 \Rx:=11.4, \Ry:=-15, \Rz:=0), v200, z200, Tooldata_7;
MoveJ RelTool (starting_position, 48, 246.4, -457 \Rx:=10.9, \Ry:=-15, \Rz:=0), v200, z200, Tooldata_7;
MoveJ RelTool (starting_position, 49, 247, -455 \Rx:=10.4, \Ry:=-14.7, \Rz:=0), v200, z200, Tooldata_7;
MoveJ RelTool (starting_position, 51, 247.6, -452 \Rx:=9.8, \Ry:=-14.4, \Rz:=0), v200, z200, Tooldata_7;
MoveJ RelTool (starting_position, 53, 248.2, -450 \Rx:=9.2, \Ry:=-14.1, \Rz:=0), v200, z200, Tooldata_7;
MoveJ RelTool (starting_position, 55, 248.8, -449 \Rx:=8.5, \Ry:=-13.8, \Rz:=0), v200, z200, Tooldata_7;
MoveJ RelTool (starting_position, 57, 249.5, -447 \Rx:=7.9, \Ry:=-13.2, \Rz:=0), v200, z200, Tooldata_7;
MoveJ RelTool (starting_position, 59, 250.2, -445 \Rx:=7.3, \Ry:=-12.9, \Rz:=0), v200, z200, Tooldata_7;
MoveJ RelTool (starting_position, 62, 250.9, -443 \Rx:=6.7, \Ry:=-12.6, \Rz:=0), v200, z200, Tooldata_7;
MoveJ RelTool (starting_position, 64, 251.6, -442 \Rx:=6.1, \Ry:=-12, \Rz:=0), v200, z200, Tooldata_7;
MoveJ RelTool (starting_position, 67, 252.4, -440 \Rx:=5.5, \Ry:=-11.7, \Rz:=0), v200, z200, Tooldata_7;
MoveJ RelTool (starting_position, 70, 253.1, -439 \Rx:=4.8, \Ry:=-11.1, \Rz:=0), v200, z200, Tooldata_7;
MoveJ RelTool (starting_position, 73, 253.8, -438 \Rx:=4.2, \Ry:=-10.5, \Rz:=0), v200, z200, Tooldata_7;
MoveJ RelTool (starting_position, 76, 254.6, -437 \Rx:=3.6, \Ry:=-9.9, \Rz:=0), v200, z200, Tooldata_7;
MoveJ RelTool (starting_position, 78, 255.4, -436 \Rx:=3.1, \Ry:=-9.6, \Rz:=0), v200, z200, Tooldata_7;
MoveJ RelTool (starting_position, 81, 256.1, -435 \Rx:=2.7, \Ry:=-9, \Rz:=0), v200, z200, Tooldata_7;
MoveJ RelTool (starting_position, 83, 256.9, -434 \Rx:=2.2, \Ry:=-8.7, \Rz:=0), v200, z200, Tooldata_7;
MoveJ RelTool (starting_position, 86, 257.6, -433 \Rx:=1.9, \Ry:=-8.4, \Rz:=0), v200, z200, Tooldata_7;
MoveJ RelTool (starting_position, 88, 258.3, -433 \Rx:=1.6, \Ry:=-7.8, \Rz:=0), v200, z200, Tooldata_7;
MoveJ RelTool (starting_position, 90, 259.1, -432 \Rx:=1.2, \Ry:=-7.5, \Rz:=0), v200, z200, Tooldata_7;
MoveJ RelTool (starting_position, 92, 259.8, -432 \Rx:=1, \Ry:=-7.2, \Rz:=0), v200, z200, Tooldata_7;
MoveJ RelTool (starting_position, 94, 260.5, -431 \Rx:=0.8, \Ry:=-6.9, \Rz:=0), v200, z200, Tooldata_7;
MoveJ RelTool (starting_position, 96, 261.1, -431 \Rx:=0.6, \Ry:=-6.6, \Rz:=0), v200, z200, Tooldata_7;
MoveJ RelTool (starting_position, 97, 261.8, -431 \Rx:=0.5, \Ry:=-6.3, \Rz:=0), v200, z200, Tooldata_7;
MoveJ RelTool (starting_position, 99, 262.4, -431 \Rx:=0.5, \Ry:=-6, \Rz:=0), v200, z200, Tooldata_7;
MoveJ RelTool (starting_position, 101, 263, -431 \Rx:=0.5, \Ry:=-5.7, \Rz:=0), v200, z200, Tooldata_7;
MoveJ RelTool (starting_position, 102, 263.6, -431 \Rx:=0.5, \Ry:=-5.4, \Rz:=0), v200, z200, Tooldata_7;
MoveJ RelTool (starting_position, 103, 264.1, -431 \Rx:=0.6, \Ry:=-5.1, \Rz:=0), v200, z200, Tooldata_7;
MoveJ RelTool (starting_position, 104, 264.6, -431 \Rx:=0.7, \Ry:=-5.1, \Rz:=0), v200, z200, Tooldata_7;
MoveJ RelTool (starting_position, 104, 265.1, -431 \Rx:=0.9, \Ry:=-5.1, \Rz:=0), v200, z200, Tooldata_7;
MoveJ RelTool (starting_position, 103, 265.6, -431 \Rx:=1.1, \Ry:=-5.1, \Rz:=0), v200, z200, Tooldata_7;
MoveJ RelTool (starting_position, 103, 266, -431 \Rx:=1.2, \Ry:=-5.4, \Rz:=0), v200, z200, Tooldata_7;
MoveJ RelTool (starting_position, 102, 266.4, -431 \Rx:=1.5, \Ry:=-5.4, \Rz:=0), v200, z200, Tooldata_7;
MoveJ RelTool (starting_position, 101, 266.8, -431 \Rx:=1.7, \Ry:=-5.7, \Rz:=0), v200, z200, Tooldata_7;
MoveJ RelTool (starting_position, 100, 267.1, -431 \Rx:=1.9, \Ry:=-5.7, \Rz:=0), v200, z200, Tooldata_7;
MoveJ RelTool (starting_position, 99, 267.5, -431 \Rx:=2.2, \Ry:=-6, \Rz:=0), v200, z200, Tooldata_7;
MoveJ RelTool (starting_position, 97, 267.7, -431 \Rx:=2.5, \Ry:=-6.3, \Rz:=0), v200, z200, Tooldata_7;
MoveJ RelTool (starting_position, 96, 268, -430 \Rx:=2.9, \Ry:=-6.6, \Rz:=0), v200, z200, Tooldata_7;
MoveJ RelTool (starting_position, 94, 268.3, -430 \Rx:=3.1, \Ry:=-6.9, \Rz:=0), v200, z200, Tooldata_7;
MoveJ RelTool (starting_position, 92, 268.5, -430 \Rx:=3.4, \Ry:=-7.2, \Rz:=0), v200, z200, Tooldata_7;
MoveJ RelTool (starting_position, 89, 268.7, -429 \Rx:=3.6, \Ry:=-7.8, \Rz:=0), v200, z200, Tooldata_7;
MoveJ RelTool (starting_position, 87, 268.9, -428 \Rx:=3.8, \Ry:=-8.1, \Rz:=0), v200, z200, Tooldata_7;
MoveJ RelTool (starting_position, 85, 269, -427 \Rx:=4, \Ry:=-8.4, \Rz:=0), v200, z200, Tooldata_7;
MoveJ RelTool (starting_position, 83, 269.2, -427 \Rx:=4.1, \Ry:=-9, \Rz:=0), v200, z200, Tooldata_7;
MoveJ RelTool (starting_position, 80, 269.3, -426 \Rx:=4.3, \Ry:=-9.3, \Rz:=0), v200, z200, Tooldata_7;
MoveJ RelTool (starting_position, 78, 269.4, -424 \Rx:=4.4, \Ry:=-9.6, \Rz:=0), v200, z200, Tooldata_7;
MoveJ RelTool (starting_position, 76, 269.5, -423 \Rx:=4.6, \Ry:=-9.9, \Rz:=0), v200, z200, Tooldata_7;
MoveJ RelTool (starting_position, 75, 269.6, -422 \Rx:=4.7, \Ry:=-10.5, \Rz:=0), v200, z200, Tooldata_7;
MoveJ RelTool (starting_position, 73, 269.7, -421 \Rx:=4.8, \Ry:=-10.5, \Rz:=0), v200, z200, Tooldata_7;
MoveJ RelTool (starting_position, 71, 269.8, -419 \Rx:=4.8, \Ry:=-10.8, \Rz:=0), v200, z200, Tooldata_7;
MoveJ RelTool (starting_position, 70, 269.8, -418 \Rx:=4.9, \Ry:=-11.1, \Rz:=0), v200, z200, Tooldata_7;
MoveJ RelTool (starting_position, 68, 269.9, -416 \Rx:=5, \Ry:=-11.4, \Rz:=0), v200, z200, Tooldata_7;
MoveJ RelTool (starting_position, 67, 269.9, -415 \Rx:=5.1, \Ry:=-11.7, \Rz:=0), v200, z200, Tooldata_7;
MoveJ RelTool (starting_position, 65, 270, -413 \Rx:=5.2, \Ry:=-12, \Rz:=0), v200, z200, Tooldata_7;
MoveJ RelTool (starting_position, 64, 270, -411 \Rx:=5.4, \Ry:=-12, \Rz:=0), v200, z200, Tooldata_7;
MoveJ RelTool (starting_position, 63, 270, -410 \Rx:=5.5, \Ry:=-12.3, \Rz:=0), v200, z200, Tooldata_7;
MoveJ RelTool (starting_position, 61, 270, -408 \Rx:=5.6, \Ry:=-12.6, \Rz:=0), v200, z200, Tooldata_7;
MoveJ RelTool (starting_position, 60, 270, -407 \Rx:=5.8, \Ry:=-12.9, \Rz:=0), v200, z200, Tooldata_7;
MoveJ RelTool (starting_position, 60, 270, -405 \Rx:=5.9, \Ry:=-12.9, \Rz:=0), v200, z200, Tooldata_7;
MoveJ RelTool (starting_position, 59, 270, -403 \Rx:=6.1, \Ry:=-12.9, \Rz:=0), v200, z200, Tooldata_7;
MoveJ RelTool (starting_position, 58, 270, -402 \Rx:=6.4, \Ry:=-13.2, \Rz:=0), v200, z200, Tooldata_7;
MoveJ RelTool (starting_position, 58, 270, -400 \Rx:=6.6, \Ry:=-13.2, \Rz:=0), v200, z200, Tooldata_7;
MoveJ RelTool (starting_position, 58, 270, -398 \Rx:=6.9, \Ry:=-13.2, \Rz:=0), v200, z200, Tooldata_7;
MoveJ RelTool (starting_position, 58, 270, -397 \Rx:=7.1, \Ry:=-13.2, \Rz:=0), v200, z200, Tooldata_7;
MoveJ RelTool (starting_position, 58, 270, -395 \Rx:=7.3, \Ry:=-13.2, \Rz:=0), v200, z200, Tooldata_7;
MoveJ RelTool (starting_position, 58, 270, -394 \Rx:=7.6, \Ry:=-13.2, \Rz:=0), v200, z200, Tooldata_7;
MoveJ RelTool (starting_position, 57, 270, -392 \Rx:=7.7, \Ry:=-13.2, \Rz:=0), v200, z200, Tooldata_7;
MoveJ RelTool (starting_position, 57, 270, -391 \Rx:=7.9, \Ry:=-13.2, \Rz:=0), v200, z200, Tooldata_7;
MoveJ RelTool (starting_position, 57, 270, -390 \Rx:=8, \Ry:=-13.2, \Rz:=0), v200, z200, Tooldata_7;
MoveJ RelTool (starting_position, 56, 270, -388 \Rx:=8, \Ry:=-13.5, \Rz:=0), v200, z200, Tooldata_7;
MoveJ RelTool (starting_position, 56, 270, -387 \Rx:=8, \Ry:=-13.5, \Rz:=0), v200, z200, Tooldata_7;
MoveJ RelTool (starting_position, 55, 270, -386 \Rx:=7.9, \Ry:=-13.5, \Rz:=0), v200, z200, Tooldata_7;
MoveJ RelTool (starting_position, 55, 270, -385 \Rx:=7.8, \Ry:=-13.8, \Rz:=0), v200, z200, Tooldata_7;
MoveJ RelTool (starting_position, 54, 270, -383 \Rx:=7.6, \Ry:=-13.8, \Rz:=0), v200, z200, Tooldata_7;
MoveJ RelTool (starting_position, 54, 270, -382 \Rx:=7.3, \Ry:=-13.8, \Rz:=0), v200, z200, Tooldata_7;
MoveJ RelTool (starting_position, 53, 270, -381 \Rx:=6.9, \Ry:=-14.1, \Rz:=0), v200, z200, Tooldata_7;
MoveJ RelTool (starting_position, 52, 270, -380 \Rx:=6.5, \Ry:=-14.1, \Rz:=0), v200, z200, Tooldata_7;
MoveJ RelTool (starting_position, 52, 270, -379 \Rx:=6.1, \Ry:=-14.1, \Rz:=0), v200, z200, Tooldata_7;
MoveJ RelTool (starting_position, 51, 270, -378 \Rx:=5.5, \Ry:=-14.4, \Rz:=0), v200, z200, Tooldata_7;
MoveJ RelTool (starting_position, 50, 270, -377 \Rx:=5, \Ry:=-14.4, \Rz:=0), v200, z200, Tooldata_7;
MoveJ RelTool (starting_position, 48, 270, -376 \Rx:=4.4, \Ry:=-14.7, \Rz:=0), v200, z200, Tooldata_7;
MoveJ RelTool (starting_position, 47, 270, -375 \Rx:=3.8, \Ry:=-15, \Rz:=0), v200, z200, Tooldata_7;
MoveJ RelTool (starting_position, 45, 270, -374 \Rx:=3.2, \Ry:=-15.3, \Rz:=0), v200, z200, Tooldata_7;
MoveJ RelTool (starting_position, 43, 270, -373 \Rx:=2.5, \Ry:=-15.6, \Rz:=0), v200, z200, Tooldata_7;
MoveJ RelTool (starting_position, 41, 270, -371 \Rx:=1.8, \Ry:=-16.2, \Rz:=0), v200, z200, Tooldata_7;
MoveJ RelTool (starting_position, 39, 270, -370 \Rx:=1.1, \Ry:=-16.5, \Rz:=0), v200, z200, Tooldata_7;
MoveJ RelTool (starting_position, 37, 270, -369 \Rx:=0.5, \Ry:=-16.8, \Rz:=0), v200, z200, Tooldata_7;
MoveJ RelTool (starting_position, 35, 270, -368 \Rx:=-0.1, \Ry:=-17.1, \Rz:=0), v200, z200, Tooldata_7;
MoveJ RelTool (starting_position, 33, 270, -366 \Rx:=-0.5, \Ry:=-17.4, \Rz:=0), v200, z200, Tooldata_7;
MoveJ RelTool (starting_position, 30, 270, -365 \Rx:=-1, \Ry:=-18, \Rz:=0), v200, z200, Tooldata_7;
MoveJ RelTool (starting_position, 27, 270, -363 \Rx:=-1.4, \Ry:=-18.3, \Rz:=0), v200, z200, Tooldata_7;
MoveJ RelTool (starting_position, 25, 270, -362 \Rx:=-1.8, \Ry:=-18.9, \Rz:=0), v200, z200, Tooldata_7;
MoveJ RelTool (starting_position, 22, 270, -360 \Rx:=-2.1, \Ry:=-19.5, \Rz:=0), v200, z200, Tooldata_7;
MoveJ RelTool (starting_position, 19, 270, -358 \Rx:=-2.3, \Ry:=-19.8, \Rz:=0), v200, z200, Tooldata_7;
MoveJ RelTool (starting_position, 16, 270, -356 \Rx:=-2.5, \Ry:=-20.4, \Rz:=0), v200, z200, Tooldata_7;
MoveJ RelTool (starting_position, 13, 270, -354 \Rx:=-2.6, \Ry:=-21, \Rz:=0), v200, z200, Tooldata_7;
MoveJ RelTool (starting_position, 11, 270, -352 \Rx:=-2.6, \Ry:=-21.3, \Rz:=0), v200, z200, Tooldata_7;
MoveJ RelTool (starting_position, 8, 270, -349 \Rx:=-2.7, \Ry:=-21.9, \Rz:=0), v200, z200, Tooldata_7;
MoveJ RelTool (starting_position, 5, 270, -347 \Rx:=-2.7, \Ry:=-22.2, \Rz:=0), v200, z200, Tooldata_7;
MoveJ RelTool (starting_position, 3, 270, -344 \Rx:=-2.7, \Ry:=-22.8, \Rz:=0), v200, z200, Tooldata_7;
MoveJ RelTool (starting_position, 0, 270, -341 \Rx:=-2.6, \Ry:=-23.1, \Rz:=0), v200, z200, Tooldata_7;
MoveJ RelTool (starting_position, -2, 270, -339 \Rx:=-2.5, \Ry:=-23.7, \Rz:=0), v200, z200, Tooldata_7;
MoveJ RelTool (starting_position, -4, 270, -336 \Rx:=-2.3, \Ry:=-24, \Rz:=0), v200, z200, Tooldata_7;
MoveJ RelTool (starting_position, -7, 270, -333 \Rx:=-2.2, \Ry:=-24.3, \Rz:=0), v200, z200, Tooldata_7;
MoveJ RelTool (starting_position, -8, 270, -330 \Rx:=-2.1, \Ry:=-24.9, \Rz:=0), v200, z200, Tooldata_7;
MoveJ RelTool (starting_position, -10, 270, -327 \Rx:=-1.9, \Ry:=-24.9, \Rz:=0), v200, z200, Tooldata_7;
MoveJ RelTool (starting_position, -11, 270, -324 \Rx:=-1.8, \Ry:=-25.2, \Rz:=0), v200, z200, Tooldata_7;
MoveJ RelTool (starting_position, -13, 270, -321 \Rx:=-1.6, \Ry:=-25.5, \Rz:=0), v200, z200, Tooldata_7;
MoveJ RelTool (starting_position, -14, 270, -318 \Rx:=-1.5, \Ry:=-25.5, \Rz:=0), v200, z200, Tooldata_7;
MoveJ RelTool (starting_position, -14, 270, -315 \Rx:=-1.4, \Ry:=-25.8, \Rz:=0), v200, z200, Tooldata_7;
MoveJ RelTool (starting_position, -15, 270, -312 \Rx:=-1.2, \Ry:=-25.8, \Rz:=0), v200, z200, Tooldata_7;
MoveJ RelTool (starting_position, -16, 270, -309 \Rx:=-1.1, \Ry:=-25.8, \Rz:=0), v200, z200, Tooldata_7;
MoveJ RelTool (starting_position, -16, 270, -306 \Rx:=-1.1, \Ry:=-26.1, \Rz:=0), v200, z200, Tooldata_7;
MoveJ RelTool (starting_position, -16, 270, -303 \Rx:=-0.9, \Ry:=-26.1, \Rz:=0), v200, z200, Tooldata_7;
MoveJ RelTool (starting_position, -17, 270, -300 \Rx:=-0.8, \Ry:=-26.1, \Rz:=0), v200, z200, Tooldata_7;
MoveJ RelTool (starting_position, -16, 270, -297 \Rx:=-0.7, \Ry:=-26.1, \Rz:=0), v200, z200, Tooldata_7;
MoveJ RelTool (starting_position, -16, 270, -294 \Rx:=-0.5, \Ry:=-26.1, \Rz:=0), v200, z200, Tooldata_7;
MoveJ RelTool (starting_position, -15, 270, -291 \Rx:=-0.4, \Ry:=-25.8, \Rz:=0), v200, z200, Tooldata_7;
MoveJ RelTool (starting_position, -15, 270.1, -289 \Rx:=-0.2, \Ry:=-25.8, \Rz:=0), v200, z200, Tooldata_7;
MoveJ RelTool (starting_position, -14, 270.1, -286 \Rx:=-0.1, \Ry:=-25.5, \Rz:=0), v200, z200, Tooldata_7;
MoveJ RelTool (starting_position, -13, 270.2, -283 \Rx:=0.2, \Ry:=-25.5, \Rz:=0), v200, z200, Tooldata_7;
MoveJ RelTool (starting_position, -13, 270.3, -281 \Rx:=0.4, \Ry:=-25.5, \Rz:=0), v200, z200, Tooldata_7;
MoveJ RelTool (starting_position, -12, 270.3, -278 \Rx:=0.6, \Ry:=-25.2, \Rz:=0), v200, z200, Tooldata_7;
MoveJ RelTool (starting_position, -11, 270.4, -276 \Rx:=0.9, \Ry:=-25.2, \Rz:=0), v200, z200, Tooldata_7;
MoveJ RelTool (starting_position, -10, 270.5, -273 \Rx:=1.2, \Ry:=-24.9, \Rz:=0), v200, z200, Tooldata_7;
MoveJ RelTool (starting_position, -9, 270.7, -271 \Rx:=1.6, \Ry:=-24.6, \Rz:=0), v200, z200, Tooldata_7;
MoveJ RelTool (starting_position, -8, 270.8, -268 \Rx:=1.9, \Ry:=-24.6, \Rz:=0), v200, z200, Tooldata_7;
MoveJ RelTool (starting_position, -7, 270.9, -266 \Rx:=2.3, \Ry:=-24.3, \Rz:=0), v200, z200, Tooldata_7;
MoveJ RelTool (starting_position, -6, 271.1, -263 \Rx:=2.8, \Ry:=-24.3, \Rz:=0), v200, z200, Tooldata_7;
MoveJ RelTool (starting_position, -4, 271.3, -261 \Rx:=3.2, \Ry:=-24, \Rz:=0), v200, z200, Tooldata_7;
MoveJ RelTool (starting_position, -3, 271.5, -258 \Rx:=3.7, \Ry:=-23.7, \Rz:=0), v200, z200, Tooldata_7;
MoveJ RelTool (starting_position, -1, 271.7, -256 \Rx:=4.1, \Ry:=-23.4, \Rz:=0), v200, z200, Tooldata_7;
MoveJ RelTool (starting_position, 0, 271.9, -253 \Rx:=4.6, \Ry:=-23.1, \Rz:=0), v200, z200, Tooldata_7;
MoveJ RelTool (starting_position, 2, 272.2, -250 \Rx:=5.1, \Ry:=-22.8, \Rz:=0), v200, z200, Tooldata_7;
MoveJ RelTool (starting_position, 3, 272.5, -248 \Rx:=5.6, \Ry:=-22.8, \Rz:=0), v200, z200, Tooldata_7;
MoveJ RelTool (starting_position, 5, 272.8, -245 \Rx:=6.1, \Ry:=-22.2, \Rz:=0), v200, z200, Tooldata_7;
MoveJ RelTool (starting_position, 7, 273.2, -243 \Rx:=6.6, \Ry:=-21.9, \Rz:=0), v200, z200, Tooldata_7;
MoveJ RelTool (starting_position, 9, 273.6, -240 \Rx:=7, \Ry:=-21.6, \Rz:=0), v200, z200, Tooldata_7;
MoveJ RelTool (starting_position, 11, 274, -237 \Rx:=7.4, \Ry:=-21.3, \Rz:=0), v200, z200, Tooldata_7;
MoveJ RelTool (starting_position, 12, 274.4, -235 \Rx:=7.8, \Ry:=-21, \Rz:=0), v200, z200, Tooldata_7;
MoveJ RelTool (starting_position, 14, 274.8, -232 \Rx:=8.2, \Ry:=-20.7, \Rz:=0), v200, z200, Tooldata_7;
MoveJ RelTool (starting_position, 16, 275.3, -230 \Rx:=8.6, \Ry:=-20.4, \Rz:=0), v200, z200, Tooldata_7;
MoveJ RelTool (starting_position, 18, 275.9, -228 \Rx:=8.9, \Ry:=-20.1, \Rz:=0), v200, z200, Tooldata_7;
MoveJ RelTool (starting_position, 20, 276.4, -225 \Rx:=9.2, \Ry:=-19.8, \Rz:=0), v200, z200, Tooldata_7;
MoveJ RelTool (starting_position, 21, 277, -223 \Rx:=9.5, \Ry:=-19.5, \Rz:=0), v200, z200, Tooldata_7;
MoveJ RelTool (starting_position, 24, 277.6, -221 \Rx:=9.7, \Ry:=-19.2, \Rz:=0), v200, z200, Tooldata_7;
MoveJ RelTool (starting_position, 26, 278.2, -219 \Rx:=10, \Ry:=-18.6, \Rz:=0), v200, z200, Tooldata_7;
MoveJ RelTool (starting_position, 28, 278.8, -217 \Rx:=10.2, \Ry:=-18.3, \Rz:=0), v200, z200, Tooldata_7;
MoveJ RelTool (starting_position, 30, 279.5, -215 \Rx:=10.4, \Ry:=-18, \Rz:=0), v200, z200, Tooldata_7;
MoveJ RelTool (starting_position, 33, 280.2, -214 \Rx:=10.6, \Ry:=-17.4, \Rz:=0), v200, z200, Tooldata_7;
MoveJ RelTool (starting_position, 35, 280.9, -212 \Rx:=10.8, \Ry:=-17.1, \Rz:=0), v200, z200, Tooldata_7;
MoveJ RelTool (starting_position, 37, 281.6, -210 \Rx:=10.9, \Ry:=-16.8, \Rz:=0), v200, z200, Tooldata_7;
MoveJ RelTool (starting_position, 40, 282.4, -209 \Rx:=11, \Ry:=-16.2, \Rz:=0), v200, z200, Tooldata_7;
MoveJ RelTool (starting_position, 42, 283.1, -207 \Rx:=11.1, \Ry:=-15.9, \Rz:=0), v200, z200, Tooldata_7;
MoveJ RelTool (starting_position, 44, 283.8, -206 \Rx:=11.2, \Ry:=-15.6, \Rz:=0), v200, z200, Tooldata_7;
MoveJ RelTool (starting_position, 47, 284.6, -204 \Rx:=11.2, \Ry:=-15, \Rz:=0), v200, z200, Tooldata_7;
MoveJ RelTool (starting_position, 49, 285.4, -203 \Rx:=11.2, \Ry:=-14.7, \Rz:=0), v200, z200, Tooldata_7;
MoveJ RelTool (starting_position, 52, 286.1, -201 \Rx:=11.2, \Ry:=-14.1, \Rz:=0), v200, z200, Tooldata_7;
MoveJ RelTool (starting_position, 55, 286.9, -200 \Rx:=11.2, \Ry:=-13.8, \Rz:=0), v200, z200, Tooldata_7;
MoveJ RelTool (starting_position, 57, 287.6, -198 \Rx:=11.2, \Ry:=-13.2, \Rz:=0), v200, z200, Tooldata_7;
MoveJ RelTool (starting_position, 60, 288.3, -197 \Rx:=11.2, \Ry:=-12.6, \Rz:=0), v200, z200, Tooldata_7;
MoveJ RelTool (starting_position, 63, 289.1, -195 \Rx:=11.1, \Ry:=-12.3, \Rz:=0), v200, z200, Tooldata_7;
MoveJ RelTool (starting_position, 66, 289.8, -194 \Rx:=11.1, \Ry:=-11.7, \Rz:=0), v200, z200, Tooldata_7;
MoveJ RelTool (starting_position, 70, 290.5, -193 \Rx:=10.9, \Ry:=-11.1, \Rz:=0), v200, z200, Tooldata_7;
MoveJ RelTool (starting_position, 73, 291.1, -191 \Rx:=10.8, \Ry:=-10.5, \Rz:=0), v200, z200, Tooldata_7;
MoveJ RelTool (starting_position, 76, 291.8, -190 \Rx:=10.6, \Ry:=-9.9, \Rz:=0), v200, z200, Tooldata_7;
MoveJ RelTool (starting_position, 79, 292.4, -189 \Rx:=10.5, \Ry:=-9.6, \Rz:=0), v200, z200, Tooldata_7;
MoveJ RelTool (starting_position, 82, 293, -187 \Rx:=10.3, \Ry:=-9, \Rz:=0), v200, z200, Tooldata_7;
MoveJ RelTool (starting_position, 86, 293.6, -186 \Rx:=10.2, \Ry:=-8.4, \Rz:=0), v200, z200, Tooldata_7;
MoveJ RelTool (starting_position, 89, 294.1, -185 \Rx:=10, \Ry:=-7.8, \Rz:=0), v200, z200, Tooldata_7;
MoveJ RelTool (starting_position, 94, 294.6, -183 \Rx:=9.8, \Ry:=-6.9, \Rz:=0), v200, z200, Tooldata_7;
MoveJ RelTool (starting_position, 98, 295.1, -182 \Rx:=9.6, \Ry:=-6.3, \Rz:=0), v200, z200, Tooldata_7;
MoveJ RelTool (starting_position, 102, 295.6, -181 \Rx:=9.3, \Ry:=-5.4, \Rz:=0), v200, z200, Tooldata_7;
MoveJ RelTool (starting_position, 106, 296, -180 \Rx:=9.1, \Ry:=-4.8, \Rz:=0), v200, z200, Tooldata_7;
MoveJ RelTool (starting_position, 111, 296.4, -179 \Rx:=8.8, \Ry:=-3.9, \Rz:=0), v200, z200, Tooldata_7;
MoveJ RelTool (starting_position, 115, 296.8, -178 \Rx:=8.5, \Ry:=-3.3, \Rz:=0), v200, z200, Tooldata_7;
MoveJ RelTool (starting_position, 119, 297.1, -178 \Rx:=8.2, \Ry:=-2.4, \Rz:=0), v200, z200, Tooldata_7;
MoveJ RelTool (starting_position, 124, 297.5, -177 \Rx:=7.9, \Ry:=-1.8, \Rz:=0), v200, z200, Tooldata_7;
MoveJ RelTool (starting_position, 128, 297.7, -177 \Rx:=7.6, \Ry:=-0.9, \Rz:=0), v200, z200, Tooldata_7;
MoveJ RelTool (starting_position, 133, 298, -176 \Rx:=7.3, \Ry:=-0, \Rz:=0), v200, z200, Tooldata_7;
MoveJ RelTool (starting_position, 137, 298.3, -176 \Rx:=7, \Ry:=0.6, \Rz:=0), v200, z200, Tooldata_7;
MoveJ RelTool (starting_position, 141, 298.5, -176 \Rx:=6.7, \Ry:=1.5, \Rz:=0), v200, z200, Tooldata_7;
MoveJ RelTool (starting_position, 145, 298.7, -177 \Rx:=6.4, \Ry:=2.1, \Rz:=0), v200, z200, Tooldata_7;
MoveJ RelTool (starting_position, 149, 298.9, -177 \Rx:=6, \Ry:=2.7, \Rz:=0), v200, z200, Tooldata_7;
MoveJ RelTool (starting_position, 152, 299, -178 \Rx:=5.7, \Ry:=3.3, \Rz:=0), v200, z200, Tooldata_7;
MoveJ RelTool (starting_position, 155, 299.2, -178 \Rx:=5.4, \Ry:=3.6, \Rz:=0), v200, z200, Tooldata_7;
MoveJ RelTool (starting_position, 158, 299.3, -179 \Rx:=5, \Ry:=4.2, \Rz:=0), v200, z200, Tooldata_7;
MoveJ RelTool (starting_position, 161, 299.4, -180 \Rx:=4.7, \Ry:=4.8, \Rz:=0), v200, z200, Tooldata_7;
MoveJ RelTool (starting_position, 163, 299.5, -181 \Rx:=4.4, \Ry:=5.1, \Rz:=0), v200, z200, Tooldata_7;
MoveJ RelTool (starting_position, 165, 299.6, -182 \Rx:=4.2, \Ry:=5.7, \Rz:=0), v200, z200, Tooldata_7;
MoveJ RelTool (starting_position, 167, 299.7, -184 \Rx:=3.9, \Ry:=6, \Rz:=0), v200, z200, Tooldata_7;
MoveJ RelTool (starting_position, 169, 299.8, -185 \Rx:=3.6, \Ry:=6, \Rz:=0), v200, z200, Tooldata_7;
MoveJ RelTool (starting_position, 170, 299.8, -187 \Rx:=3.3, \Ry:=6.3, \Rz:=0), v200, z200, Tooldata_7;
MoveJ RelTool (starting_position, 171, 299.9, -188 \Rx:=3.1, \Ry:=6.6, \Rz:=0), v200, z200, Tooldata_7;
MoveJ RelTool (starting_position, 171, 299.9, -190 \Rx:=2.9, \Ry:=6.6, \Rz:=0), v200, z200, Tooldata_7;
MoveJ RelTool (starting_position, 171, 300, -191 \Rx:=2.7, \Ry:=6.6, \Rz:=0), v200, z200, Tooldata_7;
MoveJ RelTool (starting_position, 171, 300, -193 \Rx:=2.6, \Ry:=6.6, \Rz:=0), v200, z200, Tooldata_7;
MoveJ RelTool (starting_position, 171, 300, -194 \Rx:=2.6, \Ry:=6.6, \Rz:=0), v200, z200, Tooldata_7;
MoveJ RelTool (starting_position, 170, 300, -196 \Rx:=2.6, \Ry:=6.3, \Rz:=0), v200, z200, Tooldata_7;
MoveJ RelTool (starting_position, 169, 300, -197 \Rx:=2.7, \Ry:=6.3, \Rz:=0), v200, z200, Tooldata_7;
MoveJ RelTool (starting_position, 168, 300, -199 \Rx:=2.8, \Ry:=6, \Rz:=0), v200, z200, Tooldata_7;
MoveJ RelTool (starting_position, 166, 300, -200 \Rx:=2.9, \Ry:=5.7, \Rz:=0), v200, z200, Tooldata_7;
MoveJ RelTool (starting_position, 165, 300, -201 \Rx:=3.1, \Ry:=5.4, \Rz:=0), v200, z200, Tooldata_7;
MoveJ RelTool (starting_position, 163, 300, -202 \Rx:=3.4, \Ry:=5.1, \Rz:=0), v200, z200, Tooldata_7;
MoveJ RelTool (starting_position, 161, 300, -203 \Rx:=3.7, \Ry:=4.8, \Rz:=0), v200, z200, Tooldata_7;
MoveJ RelTool (starting_position, 158, 300, -203 \Rx:=4, \Ry:=4.2, \Rz:=0), v200, z200, Tooldata_7;
MoveJ RelTool (starting_position, 156, 300, -204 \Rx:=4.3, \Ry:=3.9, \Rz:=0), v200, z200, Tooldata_7;
MoveJ RelTool (starting_position, 153, 300, -204 \Rx:=4.6, \Ry:=3.3, \Rz:=0), v200, z200, Tooldata_7;
MoveJ RelTool (starting_position, 150, 300, -204 \Rx:=4.8, \Ry:=3, \Rz:=0), v200, z200, Tooldata_7;
MoveJ RelTool (starting_position, 148, 300, -204 \Rx:=5.1, \Ry:=2.4, \Rz:=0), v200, z200, Tooldata_7;
MoveJ RelTool (starting_position, 145, 300, -204 \Rx:=5.4, \Ry:=1.8, \Rz:=0), v200, z200, Tooldata_7;
MoveJ RelTool (starting_position, 142, 300, -204 \Rx:=5.6, \Ry:=1.5, \Rz:=0), v200, z200, Tooldata_7;
MoveJ RelTool (starting_position, 140, 300, -204 \Rx:=5.8, \Ry:=0.9, \Rz:=0), v200, z200, Tooldata_7;
MoveJ RelTool (starting_position, 138, 300, -203 \Rx:=6, \Ry:=0.6, \Rz:=0), v200, z200, Tooldata_7;
MoveJ RelTool (starting_position, 136, 300, -203 \Rx:=6.2, \Ry:=0.3, \Rz:=0), v200, z200, Tooldata_7;
MoveJ RelTool (starting_position, 134, 300, -202 \Rx:=6.3, \Ry:=-0, \Rz:=0), v200, z200, Tooldata_7;
MoveJ RelTool (starting_position, 132, 300, -202 \Rx:=6.4, \Ry:=-0.3, \Rz:=0), v200, z200, Tooldata_7;
MoveJ RelTool (starting_position, 131, 300, -201 \Rx:=6.4, \Ry:=-0.6, \Rz:=0), v200, z200, Tooldata_7;
MoveJ RelTool (starting_position, 130, 300, -200 \Rx:=6.4, \Ry:=-0.6, \Rz:=0), v200, z200, Tooldata_7;
MoveJ RelTool (starting_position, 129, 300, -199 \Rx:=6.4, \Ry:=-0.9, \Rz:=0), v200, z200, Tooldata_7;
MoveJ RelTool (starting_position, 128, 300, -198 \Rx:=6.3, \Ry:=-1.2, \Rz:=0), v200, z200, Tooldata_7;
MoveJ RelTool (starting_position, 127, 300, -197 \Rx:=6.1, \Ry:=-1.2, \Rz:=0), v200, z200, Tooldata_7;
MoveJ RelTool (starting_position, 126, 300, -197 \Rx:=6, \Ry:=-1.5, \Rz:=0), v200, z200, Tooldata_7;
MoveJ RelTool (starting_position, 126, 300, -196 \Rx:=5.7, \Ry:=-1.5, \Rz:=0), v200, z200, Tooldata_7;
MoveJ RelTool (starting_position, 125, 300, -195 \Rx:=5.6, \Ry:=-1.5, \Rz:=0), v200, z200, Tooldata_7;
MoveJ RelTool (starting_position, 125, 300, -194 \Rx:=5.3, \Ry:=-1.5, \Rz:=0), v200, z200, Tooldata_7;
MoveJ RelTool (starting_position, 126, 300, -193 \Rx:=5, \Ry:=-1.5, \Rz:=0), v200, z200, Tooldata_7;
MoveJ RelTool (starting_position, 126, 300, -193 \Rx:=4.7, \Ry:=-1.5, \Rz:=0), v200, z200, Tooldata_7;
MoveJ RelTool (starting_position, 127, 300, -192 \Rx:=4.3, \Ry:=-1.2, \Rz:=0), v200, z200, Tooldata_7;
MoveJ RelTool (starting_position, 127, 300, -192 \Rx:=3.9, \Ry:=-1.2, \Rz:=0), v200, z200, Tooldata_7;
MoveJ RelTool (starting_position, 128, 300, -191 \Rx:=3.5, \Ry:=-0.9, \Rz:=0), v200, z200, Tooldata_7;
MoveJ RelTool (starting_position, 129, 300, -191 \Rx:=3.1, \Ry:=-0.9, \Rz:=0), v200, z200, Tooldata_7;
MoveJ RelTool (starting_position, 130, 300, -191 \Rx:=2.6, \Ry:=-0.6, \Rz:=0), v200, z200, Tooldata_7;
MoveJ RelTool (starting_position, 132, 300, -191 \Rx:=2.2, \Ry:=-0.3, \Rz:=0), v200, z200, Tooldata_7;
MoveJ RelTool (starting_position, 133, 300, -191 \Rx:=1.8, \Ry:=-0, \Rz:=0), v200, z200, Tooldata_7;
MoveJ RelTool (starting_position, 134, 300, -191 \Rx:=1.5, \Ry:=0, \Rz:=0), v200, z200, Tooldata_7;
MoveJ RelTool (starting_position, 135, 300, -191 \Rx:=1.1, \Ry:=0.3, \Rz:=0), v200, z200, Tooldata_7;
MoveJ RelTool (starting_position, 136, 300, -192 \Rx:=0.8, \Ry:=0.6, \Rz:=0), v200, z200, Tooldata_7;
MoveJ RelTool (starting_position, 137, 300, -192 \Rx:=0.5, \Ry:=0.6, \Rz:=0), v200, z200, Tooldata_7;
MoveJ RelTool (starting_position, 137, 300, -192 \Rx:=0.2, \Ry:=0.6, \Rz:=0), v200, z200, Tooldata_7;
MoveJ RelTool (starting_position, 138, 300, -193 \Rx:=-0.1, \Ry:=0.6, \Rz:=0), v200, z200, Tooldata_7;
MoveJ RelTool (starting_position, 138, 300, -193 \Rx:=-0.2, \Ry:=0.9, \Rz:=0), v200, z200, Tooldata_7;
MoveJ RelTool (starting_position, 139, 300, -194 \Rx:=-0.4, \Ry:=0.9, \Rz:=0), v200, z200, Tooldata_7;
MoveJ RelTool (starting_position, 139, 300, -194 \Rx:=-0.5, \Ry:=0.9, \Rz:=0), v200, z200, Tooldata_7;
MoveJ RelTool (starting_position, 140, 300, -195 \Rx:=-0.7, \Ry:=1.2, \Rz:=0), v200, z200, Tooldata_7;
MoveJ RelTool (starting_position, 140, 300, -195 \Rx:=-0.7, \Ry:=1.2, \Rz:=0), v200, z200, Tooldata_7;
MoveJ RelTool (starting_position, 140, 300, -196 \Rx:=-0.8, \Ry:=1.2, \Rz:=0), v200, z200, Tooldata_7;
MoveJ RelTool (starting_position, 140, 300, -196 \Rx:=-0.9, \Ry:=1.2, \Rz:=0), v200, z200, Tooldata_7;
MoveJ RelTool (starting_position, 140, 300, -196 \Rx:=-0.8, \Ry:=1.2, \Rz:=0), v200, z200, Tooldata_7;
MoveJ RelTool (starting_position, 139, 300, -197 \Rx:=-0.8, \Ry:=0.9, \Rz:=0), v200, z200, Tooldata_7;
MoveJ RelTool (starting_position, 139, 300, -197 \Rx:=-0.7, \Ry:=0.9, \Rz:=0), v200, z200, Tooldata_7;
MoveJ RelTool (starting_position, 138, 300, -197 \Rx:=-0.6, \Ry:=0.9, \Rz:=0), v200, z200, Tooldata_7;
MoveJ RelTool (starting_position, 138, 300, -198 \Rx:=-0.6, \Ry:=0.6, \Rz:=0), v200, z200, Tooldata_7;
MoveJ RelTool (starting_position, 137, 300, -198 \Rx:=-0.5, \Ry:=0.6, \Rz:=0), v200, z200, Tooldata_7;
MoveJ RelTool (starting_position, 136, 300, -198 \Rx:=-0.3, \Ry:=0.6, \Rz:=0), v200, z200, Tooldata_7;
MoveJ RelTool (starting_position, 135, 300, -198 \Rx:=-0.2, \Ry:=0.3, \Rz:=0), v200, z200, Tooldata_7;
MoveJ RelTool (starting_position, 134, 300, -198 \Rx:=-0.1, \Ry:=0, \Rz:=0), v200, z200, Tooldata_7;
MoveJ RelTool (starting_position, 133, 300, -199 \Rx:=0.1, \Ry:=-0.3, \Rz:=0), v200, z200, Tooldata_7;
MoveJ RelTool (starting_position, 131, 300, -199 \Rx:=0.2, \Ry:=-0.6, \Rz:=0), v200, z200, Tooldata_7;
MoveJ RelTool (starting_position, 130, 300, -199 \Rx:=0.3, \Ry:=-0.6, \Rz:=0), v200, z200, Tooldata_7;
MoveJ RelTool (starting_position, 129, 300, -199 \Rx:=0.4, \Ry:=-0.6, \Rz:=0), v200, z200, Tooldata_7;
MoveJ RelTool (starting_position, 128, 300, -198 \Rx:=0.4, \Ry:=-0.9, \Rz:=0), v200, z200, Tooldata_7;
MoveJ RelTool (starting_position, 127, 300, -198 \Rx:=0.5, \Ry:=-1.2, \Rz:=0), v200, z200, Tooldata_7;
MoveJ RelTool (starting_position, 126, 300, -198 \Rx:=0.5, \Ry:=-1.2, \Rz:=0), v200, z200, Tooldata_7;
MoveJ RelTool (starting_position, 125, 300, -198 \Rx:=0.6, \Ry:=-1.5, \Rz:=0), v200, z200, Tooldata_7;
MoveJ RelTool (starting_position, 124, 300, -198 \Rx:=0.6, \Ry:=-1.8, \Rz:=0), v200, z200, Tooldata_7;
MoveJ RelTool (starting_position, 123, 300, -197 \Rx:=0.6, \Ry:=-1.8, \Rz:=0), v200, z200, Tooldata_7;
MoveJ RelTool (starting_position, 122, 300, -197 \Rx:=0.6, \Ry:=-2.1, \Rz:=0), v200, z200, Tooldata_7;
MoveJ RelTool (starting_position, 121, 300, -197 \Rx:=0.6, \Ry:=-2.1, \Rz:=0), v200, z200, Tooldata_7;
MoveJ RelTool (starting_position, 121, 300, -196 \Rx:=0.7, \Ry:=-2.4, \Rz:=0), v200, z200, Tooldata_7;
MoveJ RelTool (starting_position, 120, 300, -196 \Rx:=0.7, \Ry:=-2.4, \Rz:=0), v200, z200, Tooldata_7;
MoveJ RelTool (starting_position, 119, 300, -196 \Rx:=0.8, \Ry:=-2.4, \Rz:=0), v200, z200, Tooldata_7;
MoveJ RelTool (starting_position, 119, 300, -195 \Rx:=0.8, \Ry:=-2.7, \Rz:=0), v200, z200, Tooldata_7;
MoveJ RelTool (starting_position, 119, 300, -195 \Rx:=0.9, \Ry:=-2.7, \Rz:=0), v200, z200, Tooldata_7;
MoveJ RelTool (starting_position, 118, 300, -194 \Rx:=0.9, \Ry:=-2.7, \Rz:=0), v200, z200, Tooldata_7;
MoveJ RelTool (starting_position, 118, 300, -194 \Rx:=1, \Ry:=-2.7, \Rz:=0), v200, z200, Tooldata_7;
MoveJ RelTool (starting_position, 118, 300, -193 \Rx:=1, \Ry:=-2.7, \Rz:=0), v200, z200, Tooldata_7;
MoveJ RelTool (starting_position, 118, 300, -193 \Rx:=1.1, \Ry:=-2.7, \Rz:=0), v200, z200, Tooldata_7;
MoveJ RelTool (starting_position, 118, 300, -192 \Rx:=1.2, \Ry:=-2.7, \Rz:=0), v200, z200, Tooldata_7;
MoveJ RelTool (starting_position, 119, 300, -191 \Rx:=1.3, \Ry:=-2.7, \Rz:=0), v200, z200, Tooldata_7;
MoveJ RelTool (starting_position, 119, 300, -191 \Rx:=1.3, \Ry:=-2.7, \Rz:=0), v200, z200, Tooldata_7;
MoveJ RelTool (starting_position, 119, 300, -190 \Rx:=1.3, \Ry:=-2.4, \Rz:=0), v200, z200, Tooldata_7;
MoveJ RelTool (starting_position, 120, 300, -190 \Rx:=1.4, \Ry:=-2.4, \Rz:=0), v200, z200, Tooldata_7;
MoveJ RelTool (starting_position, 121, 300, -189 \Rx:=1.4, \Ry:=-2.4, \Rz:=0), v200, z200, Tooldata_7;
MoveJ RelTool (starting_position, 123, 300, -188 \Rx:=1.4, \Ry:=-2.1, \Rz:=0), v200, z200, Tooldata_7;
MoveJ RelTool (starting_position, 124, 300, -188 \Rx:=1.3, \Ry:=-1.5, \Rz:=0), v200, z200, Tooldata_7;
MoveJ RelTool (starting_position, 126, 300, -188 \Rx:=1.3, \Ry:=-1.2, \Rz:=0), v200, z200, Tooldata_7;
MoveJ RelTool (starting_position, 127, 300, -187 \Rx:=1.1, \Ry:=-1.2, \Rz:=0), v200, z200, Tooldata_7;
MoveJ RelTool (starting_position, 129, 300, -187 \Rx:=1, \Ry:=-0.9, \Rz:=0), v200, z200, Tooldata_7;
MoveJ RelTool (starting_position, 131, 300, -187 \Rx:=0.9, \Ry:=-0.6, \Rz:=0), v200, z200, Tooldata_7;
MoveJ RelTool (starting_position, 132, 300, -186 \Rx:=0.7, \Ry:=-0, \Rz:=0), v200, z200, Tooldata_7;
MoveJ RelTool (starting_position, 134, 300, -186 \Rx:=0.5, \Ry:=0, \Rz:=0), v200, z200, Tooldata_7;
MoveJ RelTool (starting_position, 136, 300, -186 \Rx:=0.3, \Ry:=0.3, \Rz:=0), v200, z200, Tooldata_7;
MoveJ RelTool (starting_position, 137, 300, -186 \Rx:=0.2, \Ry:=0.6, \Rz:=0), v200, z200, Tooldata_7;
MoveJ RelTool (starting_position, 139, 300, -186 \Rx:=-0, \Ry:=0.9, \Rz:=0), v200, z200, Tooldata_7;
MoveJ RelTool (starting_position, 140, 300, -187 \Rx:=-0.2, \Ry:=1.2, \Rz:=0), v200, z200, Tooldata_7;
MoveJ RelTool (starting_position, 141, 300, -187 \Rx:=-0.3, \Ry:=1.2, \Rz:=0), v200, z200, Tooldata_7;
MoveJ RelTool (starting_position, 143, 300, -187 \Rx:=-0.5, \Ry:=1.5, \Rz:=0), v200, z200, Tooldata_7;
MoveJ RelTool (starting_position, 144, 300, -188 \Rx:=-0.6, \Ry:=1.8, \Rz:=0), v200, z200, Tooldata_7;
MoveJ RelTool (starting_position, 146, 300, -188 \Rx:=-0.6, \Ry:=2.1, \Rz:=0), v200, z200, Tooldata_7;
MoveJ RelTool (starting_position, 147, 300, -188 \Rx:=-0.6, \Ry:=2.4, \Rz:=0), v200, z200, Tooldata_7;
MoveJ RelTool (starting_position, 149, 300, -189 \Rx:=-0.5, \Ry:=2.7, \Rz:=0), v200, z200, Tooldata_7;
MoveJ RelTool (starting_position, 150, 300, -190 \Rx:=-0.4, \Ry:=3, \Rz:=0), v200, z200, Tooldata_7;
MoveJ RelTool (starting_position, 151, 300, -190 \Rx:=-0.2, \Ry:=3, \Rz:=0), v200, z200, Tooldata_7;
MoveJ RelTool (starting_position, 152, 300, -191 \Rx:=-0, \Ry:=3.3, \Rz:=0), v200, z200, Tooldata_7;
MoveJ RelTool (starting_position, 152, 300, -192 \Rx:=0.3, \Ry:=3.3, \Rz:=0), v200, z200, Tooldata_7;
MoveJ RelTool (starting_position, 153, 300, -192 \Rx:=0.6, \Ry:=3.3, \Rz:=0), v200, z200, Tooldata_7;
MoveJ RelTool (starting_position, 153, 300, -193 \Rx:=0.9, \Ry:=3.3, \Rz:=0), v200, z200, Tooldata_7;
MoveJ RelTool (starting_position, 153, 300, -194 \Rx:=1.3, \Ry:=3.3, \Rz:=0), v200, z200, Tooldata_7;
MoveJ RelTool (starting_position, 153, 300, -195 \Rx:=1.7, \Ry:=3.3, \Rz:=0), v200, z200, Tooldata_7;
MoveJ RelTool (starting_position, 153, 300, -195 \Rx:=2.1, \Ry:=3.3, \Rz:=0), v200, z200, Tooldata_7;
MoveJ RelTool (starting_position, 152, 300, -196 \Rx:=2.5, \Ry:=3.3, \Rz:=0), v200, z200, Tooldata_7;
MoveJ RelTool (starting_position, 152, 300, -197 \Rx:=2.9, \Ry:=3.3, \Rz:=0), v200, z200, Tooldata_7;
MoveJ RelTool (starting_position, 152, 300, -197 \Rx:=3.3, \Ry:=3, \Rz:=0), v200, z200, Tooldata_7;
MoveJ RelTool (starting_position, 151, 300, -198 \Rx:=3.6, \Ry:=3, \Rz:=0), v200, z200, Tooldata_7;
MoveJ RelTool (starting_position, 151, 300, -198 \Rx:=4, \Ry:=3, \Rz:=0), v200, z200, Tooldata_7;
MoveJ RelTool (starting_position, 150, 300, -199 \Rx:=4.2, \Ry:=3, \Rz:=0), v200, z200, Tooldata_7;
MoveJ RelTool (starting_position, 150, 300, -199 \Rx:=4.4, \Ry:=2.7, \Rz:=0), v200, z200, Tooldata_7;
MoveJ RelTool (starting_position, 149, 300, -199 \Rx:=4.6, \Ry:=2.7, \Rz:=0), v200, z200, Tooldata_7;
MoveJ RelTool (starting_position, 148, 300, -200 \Rx:=4.6, \Ry:=2.4, \Rz:=0), v200, z200, Tooldata_7;
MoveJ RelTool (starting_position, 146, 300, -200 \Rx:=4.7, \Ry:=2.1, \Rz:=0), v200, z200, Tooldata_7;
MoveJ RelTool (starting_position, 145, 300, -200 \Rx:=4.6, \Ry:=2.1, \Rz:=0), v200, z200, Tooldata_7;
MoveJ RelTool (starting_position, 144, 300, -200 \Rx:=4.5, \Ry:=1.8, \Rz:=0), v200, z200, Tooldata_7;
MoveJ RelTool (starting_position, 142, 300, -200 \Rx:=4.4, \Ry:=1.5, \Rz:=0), v200, z200, Tooldata_7;
MoveJ RelTool (starting_position, 141, 300, -200 \Rx:=4.2, \Ry:=1.2, \Rz:=0), v200, z200, Tooldata_7;
MoveJ RelTool (starting_position, 139, 300, -200 \Rx:=3.9, \Ry:=0.9, \Rz:=0), v200, z200, Tooldata_7;
MoveJ RelTool (starting_position, 138, 300, -200 \Rx:=3.7, \Ry:=0.6, \Rz:=0), v200, z200, Tooldata_7;
MoveJ RelTool (starting_position, 137, 300, -200 \Rx:=3.4, \Ry:=0.6, \Rz:=0), v200, z200, Tooldata_7;
MoveJ RelTool (starting_position, 136, 300, -199 \Rx:=3, \Ry:=0.3, \Rz:=0), v200, z200, Tooldata_7;
MoveJ RelTool (starting_position, 135, 300, -199 \Rx:=2.6, \Ry:=0.3, \Rz:=0), v200, z200, Tooldata_7;
MoveJ RelTool (starting_position, 134, 300, -199 \Rx:=2.2, \Ry:=-0, \Rz:=0), v200, z200, Tooldata_7;
MoveJ RelTool (starting_position, 133, 300, -199 \Rx:=1.8, \Ry:=-0.3, \Rz:=0), v200, z200, Tooldata_7;
MoveJ RelTool (starting_position, 131, 300, -199 \Rx:=1.4, \Ry:=-0.3, \Rz:=0), v200, z200, Tooldata_7;
MoveJ RelTool (starting_position, 130, 300, -199 \Rx:=1, \Ry:=-0.6, \Rz:=0), v200, z200, Tooldata_7;
MoveJ RelTool (starting_position, 129, 300, -198 \Rx:=0.6, \Ry:=-0.9, \Rz:=0), v200, z200, Tooldata_7;
MoveJ RelTool (starting_position, 128, 300, -198 \Rx:=0.3, \Ry:=-0.9, \Rz:=0), v200, z200, Tooldata_7;
MoveJ RelTool (starting_position, 128, 300, -198 \Rx:=-0, \Ry:=-1.2, \Rz:=0), v200, z200, Tooldata_7;
MoveJ RelTool (starting_position, 127, 300, -198 \Rx:=-0.3, \Ry:=-1.2, \Rz:=0), v200, z200, Tooldata_7;
MoveJ RelTool (starting_position, 126, 300, -198 \Rx:=-0.6, \Ry:=-1.2, \Rz:=0), v200, z200, Tooldata_7;
MoveJ RelTool (starting_position, 125, 300, -198 \Rx:=-0.8, \Ry:=-1.5, \Rz:=0), v200, z200, Tooldata_7;
MoveJ RelTool (starting_position, 125, 300, -197 \Rx:=-1, \Ry:=-1.5, \Rz:=0), v200, z200, Tooldata_7;
MoveJ RelTool (starting_position, 124, 300, -197 \Rx:=-1.1, \Ry:=-1.8, \Rz:=0), v200, z200, Tooldata_7;
MoveJ RelTool (starting_position, 124, 300, -197 \Rx:=-1.2, \Ry:=-1.8, \Rz:=0), v200, z200, Tooldata_7;
MoveJ RelTool (starting_position, 124, 300, -197 \Rx:=-1.2, \Ry:=-1.8, \Rz:=0), v200, z200, Tooldata_7;
MoveJ RelTool (starting_position, 123, 300, -197 \Rx:=-1.2, \Ry:=-1.8, \Rz:=0), v200, z200, Tooldata_7;
MoveJ RelTool (starting_position, 123, 300, -197 \Rx:=-1.2, \Ry:=-1.8, \Rz:=0), v200, z200, Tooldata_7;
MoveJ RelTool (starting_position, 123, 300, -196 \Rx:=-1.1, \Ry:=-1.8, \Rz:=0), v200, z200, Tooldata_7;
MoveJ RelTool (starting_position, 123, 300, -196 \Rx:=-0.9, \Ry:=-1.8, \Rz:=0), v200, z200, Tooldata_7;
MoveJ RelTool (starting_position, 123, 300, -196 \Rx:=-0.8, \Ry:=-1.8, \Rz:=0), v200, z200, Tooldata_7;
